C09072=1097.332,62.980,442.084,176.225,15.918,152.154
C09073=1097.327,62.731,442.101,176.223,15.918,152.154
C09074=1097.321,62.481,442.117,176.221,15.918,152.155
C09075=1097.315,62.232,442.133,176.218,15.916,152.155
C09076=1097.309,61.982,442.150,176.216,15.916,152.155
C09077=1097.304,61.733,442.167,176.213,15.915,152.156
C09078=1097.298,61.483,442.183,176.211,15.914,152.156
C09079=1097.292,61.234,442.199,176.208,15.913,152.156
C09080=1097.286,60.985,442.215,176.206,15.913,152.157
C09081=1097.280,60.735,442.232,176.204,15.912,152.157
C09082=1097.275,60.486,442.248,176.201,15.911,152.158
C09083=1097.269,60.236,442.265,176.200,15.911,152.158
C09084=1097.263,59.987,442.281,176.197,15.910,152.158
C09085=1097.257,59.738,442.297,176.195,15.909,152.158
C09086=1097.251,59.488,442.313,176.192,15.909,152.159
C09087=1097.247,59.239,442.330,176.190,15.908,152.159
C09088=1097.241,58.990,442.346,176.188,15.907,152.160
C09089=1097.235,58.741,442.362,176.185,15.906,152.160
C09090=1097.229,58.491,442.379,176.183,15.905,152.160
C09091=1097.223,58.241,442.394,176.180,15.904,152.161
C09092=1097.217,57.992,442.410,176.178,15.904,152.161
C09093=1097.212,57.742,442.427,176.176,15.903,152.161
C09094=1097.206,57.493,442.444,176.173,15.902,152.161
C09095=1097.200,57.244,442.460,176.171,15.901,152.162
C09096=1097.194,56.994,442.476,176.168,15.901,152.162
C09097=1097.188,56.745,442.492,176.167,15.900,152.162
C09098=1097.183,56.496,442.508,176.164,15.900,152.163
C09099=1097.177,56.246,442.524,176.162,15.898,152.163
C09100=1097.171,55.997,442.540,176.160,15.898,152.163
C09101=1097.166,55.747,442.557,176.157,15.897,152.164
C09102=1097.160,55.498,442.573,176.155,15.896,152.164
C09103=1097.154,55.248,442.589,176.153,15.895,152.164
C09104=1097.148,54.999,442.605,176.150,15.895,152.165
C09105=1097.143,54.750,442.621,176.148,15.894,152.165
C09106=1097.137,54.501,442.637,176.146,15.893,152.165
C09107=1097.131,54.251,442.653,176.143,15.892,152.166
C09108=1097.125,54.001,442.669,176.141,15.892,152.166
C09109=1097.119,53.752,442.685,176.139,15.890,152.166
C09110=1097.114,53.502,442.702,176.137,15.890,152.167
C09111=1097.109,53.253,442.717,176.134,15.889,152.167
C09112=1097.103,53.004,442.733,176.132,15.888,152.167
C09113=1097.097,52.754,442.750,176.130,15.887,152.167
C09114=1097.091,52.505,442.766,176.127,15.886,152.168
C09115=1097.086,52.255,442.781,176.125,15.886,152.168
C09116=1097.080,52.006,442.797,176.123,15.884,152.168
C09117=1097.074,51.757,442.814,176.120,15.884,152.169
C09118=1097.069,51.507,442.829,176.119,15.884,152.169
C09119=1097.063,51.258,442.845,176.116,15.882,152.169
C09120=1097.057,51.008,442.862,176.114,15.881,152.170
C09121=1097.052,50.759,442.877,176.111,15.880,152.170
C09122=1097.046,50.510,442.893,176.109,15.880,152.170
C09123=1097.040,50.260,442.909,176.107,15.879,152.170
C09124=1097.034,50.011,442.925,176.105,15.878,152.171
C09125=1097.029,49.762,442.941,176.103,15.877,152.171
C09126=1097.023,49.512,442.956,176.100,15.876,152.171
C09127=1097.017,49.263,442.973,176.098,15.876,152.172
C09128=1097.012,49.013,442.988,176.096,15.875,152.172
C09129=1097.006,48.764,443.004,176.093,15.874,152.172
C09130=1097.001,48.514,443.020,176.091,15.873,152.172
C09131=1096.995,48.265,443.036,176.089,15.872,152.173
C09132=1096.989,47.990,443.053,176.086,15.871,152.173
C09133=1096.982,47.715,443.071,176.084,15.870,152.173
C09134=1096.977,47.442,443.089,176.082,15.869,152.174
C09135=1096.970,47.168,443.106,176.079,15.868,152.174
C09136=1096.965,46.918,443.121,176.077,15.867,152.174
C09137=1096.959,46.668,443.137,176.074,15.867,152.175
C09138=1096.954,46.419,443.153,176.073,15.866,152.175
C09139=1096.948,46.170,443.169,176.071,15.865,152.175
C09140=1096.942,45.920,443.184,176.068,15.864,152.175
C09141=1096.937,45.671,443.200,176.066,15.863,152.176
C09142=1096.931,45.421,443.216,176.063,15.862,152.176
C09143=1096.926,45.171,443.231,176.061,15.861,152.176
C09144=1096.920,44.922,443.247,176.060,15.860,152.177
C09145=1096.915,44.672,443.263,176.057,15.859,152.177
C09146=1096.909,44.423,443.279,176.055,15.858,152.177
C09147=1096.904,44.174,443.294,176.052,15.857,152.177
C09148=1096.898,43.924,443.310,176.050,15.857,152.178
C09149=1096.891,43.675,443.325,176.048,15.856,152.178
C09150=1096.886,43.426,443.341,176.046,15.855,152.178
C09151=1096.880,43.176,443.357,176.044,15.854,152.179
C09152=1096.875,42.926,443.372,176.042,15.853,152.179
C09153=1096.870,42.677,443.388,176.039,15.852,152.179
C09154=1096.863,42.428,443.403,176.037,15.851,152.179
C09155=1096.857,42.178,443.419,176.035,15.851,152.180
C09156=1096.852,41.929,443.434,176.033,15.849,152.180
C09157=1096.846,41.679,443.450,176.031,15.849,152.180
C09158=1096.840,41.430,443.465,176.028,15.848,152.181
C09159=1096.835,41.180,443.480,176.026,15.847,152.181
C09160=1096.829,40.931,443.497,176.024,15.846,152.181
C09161=1096.823,40.681,443.512,176.021,15.845,152.181
C09162=1096.817,40.432,443.527,176.020,15.844,152.182
C09163=1096.812,40.183,443.543,176.018,15.844,152.182
C09164=1096.806,39.934,443.558,176.015,15.842,152.182
C09165=1096.801,39.684,443.574,176.013,15.842,152.182
C09166=1096.794,39.434,443.589,176.011,15.841,152.183
C09167=1096.789,39.185,443.605,176.008,15.840,152.183
C09168=1096.783,38.935,443.620,176.007,15.839,152.183
C09169=1096.778,38.686,443.635,176.005,15.838,152.183
C09170=1096.772,38.436,443.650,176.002,15.837,152.184
C09171=1096.766,38.186,443.666,176.000,15.836,152.184
C09172=1096.761,37.938,443.682,175.998,15.836,152.184
C09173=1096.755,37.688,443.697,175.996,15.834,152.184
C09174=1096.749,37.438,443.712,175.994,15.834,152.185
C09175=1096.744,37.189,443.727,175.991,15.832,152.185
C09176=1096.738,36.939,443.742,175.989,15.832,152.185
C09177=1096.732,36.691,443.758,175.987,15.831,152.186
C09178=1096.726,36.441,443.773,175.985,15.830,152.186
C09179=1096.720,36.191,443.789,175.983,15.829,152.186
C09180=1096.715,35.942,443.804,175.981,15.828,152.186
C09181=1096.709,35.692,443.819,175.978,15.827,152.187
C09182=1096.704,35.443,443.834,175.976,15.826,152.187
C09183=1096.697,35.193,443.849,175.974,15.825,152.187
C09184=1096.691,34.944,443.865,175.972,15.824,152.187
C09185=1096.686,34.695,443.880,175.970,15.823,152.188
C09186=1096.680,34.445,443.895,175.968,15.823,152.188
C09187=1096.675,34.196,443.910,175.965,15.821,152.188
C09188=1096.669,33.946,443.925,175.963,15.821,152.188
C09189=1096.664,33.697,443.941,175.961,15.820,152.189
C09190=1096.657,33.447,443.955,175.959,15.819,152.189
C09191=1096.652,33.198,443.971,175.957,15.818,152.189
C09192=1096.646,32.948,443.986,175.955,15.817,152.189
C09193=1096.640,32.698,444.001,175.952,15.816,152.190
C09194=1096.634,32.449,444.016,175.950,15.815,152.190
C09195=1096.629,32.199,444.031,175.949,15.815,152.190
C09196=1096.622,31.925,444.048,175.946,15.813,152.191
C09197=1096.616,31.651,444.064,175.944,15.813,152.191
C09198=1096.610,31.377,444.081,175.941,15.811,152.191
C09199=1096.603,31.102,444.097,175.939,15.811,152.191
C09200=1096.598,30.852,444.113,175.937,15.809,152.192
C09201=1096.592,30.603,444.128,175.935,15.809,152.192
C09202=1096.586,30.354,444.143,175.933,15.808,152.192
C09203=1096.581,30.105,444.158,175.931,15.806,152.192
C09204=1096.575,29.854,444.173,175.929,15.805,152.193
C09205=1096.569,29.605,444.187,175.927,15.805,152.193
C09206=1096.564,29.355,444.203,175.924,15.803,152.193
C09207=1096.558,29.106,444.217,175.922,15.803,152.193
C09208=1096.552,28.856,444.233,175.920,15.802,152.194
C09209=1096.547,28.607,444.247,175.918,15.801,152.194
C09210=1096.540,28.358,444.262,175.916,15.800,152.194
C09211=1096.535,28.108,444.277,175.914,15.799,152.194
C09212=1096.529,27.859,444.292,175.912,15.797,152.194
C09213=1096.523,27.610,444.307,175.910,15.797,152.195
C09214=1096.518,27.360,444.321,175.908,15.796,152.195
C09215=1096.512,27.110,444.336,175.906,15.795,152.195
C09216=1096.507,26.861,444.352,175.903,15.794,152.196
C09217=1096.500,26.611,444.367,175.901,15.793,152.196
C09218=1096.495,26.362,444.381,175.899,15.793,152.196
C09219=1096.489,26.112,444.397,175.897,15.791,152.196
C09220=1096.483,25.863,444.411,175.895,15.790,152.196
C09221=1096.477,25.613,444.425,175.893,15.789,152.197
C09222=1096.471,25.364,444.440,175.891,15.788,152.197
C09223=1096.466,25.114,444.456,175.889,15.787,152.197
C09224=1096.460,24.865,444.470,175.887,15.787,152.197
C09225=1096.454,24.615,444.484,175.885,15.786,152.198
C09226=1096.449,24.366,444.500,175.882,15.785,152.198
C09227=1096.443,24.117,444.514,175.881,15.784,152.198
C09228=1096.437,23.867,444.529,175.879,15.783,152.198
C09229=1096.432,23.618,444.544,175.876,15.782,152.199
C09230=1096.425,23.367,444.559,175.874,15.781,152.199
C09231=1096.420,23.118,444.573,175.872,15.780,152.199
C09232=1096.413,22.869,444.588,175.870,15.778,152.199
C09233=1096.409,22.619,444.602,175.868,15.778,152.200
C09234=1096.403,22.370,444.617,175.866,15.777,152.200
C09235=1096.396,22.120,444.632,175.864,15.776,152.200
C09236=1096.391,21.871,444.646,175.862,15.775,152.200
C09237=1096.385,21.621,444.661,175.860,15.774,152.200
C09238=1096.380,21.372,444.676,175.858,15.773,152.201
C09239=1096.374,21.122,444.690,175.855,15.772,152.201
C09240=1096.368,20.873,444.705,175.854,15.771,152.201
C09241=1096.363,20.623,444.720,175.852,15.770,152.201
C09242=1096.357,20.374,444.734,175.850,15.769,152.202
C09243=1096.351,20.124,444.749,175.847,15.768,152.202
C09244=1096.345,19.875,444.763,175.846,15.767,152.202
C09245=1096.339,19.625,444.778,175.844,15.766,152.202
C09246=1096.334,19.376,444.793,175.841,15.765,152.202
C09247=1096.328,19.127,444.807,175.839,15.764,152.203
C09248=1096.322,18.876,444.822,175.837,15.763,152.203
C09249=1096.316,18.627,444.836,175.836,15.763,152.203
C09250=1096.311,18.378,444.850,175.833,15.761,152.204
C09251=1096.304,18.128,444.865,175.831,15.760,152.204
C09252=1096.299,17.879,444.879,175.829,15.759,152.204
C09253=1096.293,17.629,444.894,175.828,15.759,152.204
C09254=1096.288,17.379,444.908,175.825,15.757,152.204
C09255=1096.282,17.130,444.923,175.823,15.756,152.205
C09256=1096.276,16.880,444.938,175.821,15.755,152.205
C09257=1096.270,16.631,444.952,175.820,15.755,152.205
C09258=1096.264,16.382,444.966,175.817,15.753,152.205
C09259=1096.258,16.132,444.980,175.815,15.752,152.205
C09260=1096.253,15.859,444.996,175.813,15.751,152.206
C09261=1096.246,15.586,445.012,175.811,15.750,152.206
C09262=1096.240,15.313,445.028,175.809,15.750,152.206
C09263=1096.233,15.040,445.044,175.806,15.748,152.206
C09264=1096.228,14.790,445.058,175.805,15.747,152.207
C09265=1096.222,14.542,445.072,175.803,15.746,152.207
C09266=1096.216,14.291,445.086,175.800,15.745,152.207
C09267=1096.210,14.042,445.101,175.798,15.744,152.207
C09268=1096.205,13.793,445.115,175.796,15.743,152.207
C09269=1096.199,13.542,445.129,175.795,15.743,152.208
C09270=1096.193,13.293,445.144,175.792,15.741,152.208
C09271=1096.188,13.044,445.158,175.790,15.740,152.208
C09272=1096.181,12.794,445.173,175.788,15.739,152.208
C09273=1096.176,12.545,445.186,175.787,15.739,152.209
C09274=1096.170,12.295,445.200,175.784,15.737,152.209
C09275=1096.163,12.046,445.215,175.782,15.736,152.209
C09276=1096.158,11.796,445.228,175.780,15.735,152.209
C09277=1096.152,11.547,445.243,175.779,15.735,152.210
C09278=1096.146,11.297,445.257,175.776,15.733,152.210
C09279=1096.140,11.047,445.271,175.774,15.732,152.210
C09280=1096.134,10.798,445.286,175.772,15.732,152.210
C09281=1096.129,10.549,445.300,175.770,15.731,152.210
C09282=1096.123,10.299,445.314,175.768,15.729,152.211
C09283=1096.117,10.050,445.328,175.766,15.728,152.211
C09284=1096.112,9.800,445.342,175.764,15.728,152.211
C09285=1096.105,9.550,445.356,175.763,15.726,152.211
C09286=1096.099,9.301,445.370,175.760,15.725,152.211
C09287=1096.094,9.052,445.384,175.758,15.724,152.212
C09288=1096.088,8.802,445.398,175.757,15.723,152.212
C09289=1096.082,8.552,445.412,175.755,15.723,152.212
C09290=1096.076,8.303,445.427,175.752,15.721,152.212
C09291=1096.071,8.053,445.441,175.750,15.720,152.212
C09292=1096.065,7.804,445.455,175.749,15.719,152.213
C09293=1096.059,7.554,445.468,175.747,15.719,152.213
C09294=1096.053,7.305,445.483,175.744,15.717,152.213
C09295=1096.047,7.055,445.497,175.742,15.716,152.213
C09296=1096.042,6.806,445.511,175.741,15.716,152.214
C09297=1096.036,6.556,445.525,175.739,15.714,152.214
C09298=1096.030,6.306,445.539,175.737,15.714,152.214
C09299=1096.024,6.057,445.553,175.734,15.712,152.214
C09300=1096.018,5.807,445.567,175.733,15.711,152.214
C09301=1096.013,5.558,445.580,175.731,15.710,152.215
C09302=1096.007,5.308,445.594,175.729,15.710,152.215
C09303=1096.001,5.058,445.609,175.727,15.708,152.215
C09304=1095.995,4.809,445.623,175.725,15.707,152.215
C09305=1095.989,4.560,445.636,175.723,15.706,152.215
C09306=1095.984,4.310,445.650,175.721,15.705,152.216
C09307=1095.978,4.061,445.664,175.719,15.705,152.216
C09308=1095.973,3.811,445.678,175.717,15.703,152.216
C09309=1095.967,3.561,445.692,175.715,15.702,152.216
C09310=1095.960,3.312,445.706,175.714,15.701,152.216
C09311=1095.955,3.062,445.719,175.712,15.700,152.217
C09312=1095.949,2.813,445.734,175.709,15.699,152.217
C09313=1095.944,2.563,445.748,175.707,15.698,152.217
C09314=1095.938,2.314,445.761,175.705,15.697,152.217
C09315=1095.931,2.064,445.775,175.704,15.696,152.217
C09316=1095.926,1.814,445.789,175.702,15.695,152.218
C09317=1095.921,1.565,445.803,175.700,15.694,152.218
C09318=1095.915,1.315,445.817,175.698,15.693,152.218
C09319=1095.909,1.066,445.830,175.696,15.692,152.218
C09320=1095.903,0.816,445.844,175.694,15.691,152.218
C09321=1095.898,0.567,445.858,175.692,15.690,152.219
C09322=1095.892,0.317,445.872,175.690,15.688,152.219
C09323=1095.886,0.068,445.885,175.688,15.688,152.219
C09324=1095.880,-0.203,445.900,175.687,15.687,152.219
C09325=1095.873,-0.475,445.915,175.684,15.685,152.219
C09326=1095.867,-0.746,445.931,175.682,15.685,152.220
C09327=1095.861,-1.017,445.945,175.680,15.683,152.220
C09328=1095.855,-1.266,445.959,175.678,15.682,152.220
C09329=1095.850,-1.516,445.972,175.676,15.681,152.220
C09330=1095.844,-1.765,445.986,175.674,15.680,152.220
C09331=1095.839,-2.015,446.000,175.673,15.679,152.220
C09332=1095.833,-2.264,446.013,175.671,15.678,152.221
C09333=1095.827,-2.514,446.027,175.668,15.677,152.221
C09334=1095.822,-2.763,446.041,175.666,15.676,152.221
C09335=1095.815,-3.013,446.054,175.665,15.675,152.221
C09336=1095.810,-3.262,446.068,175.663,15.674,152.221
C09337=1095.804,-3.512,446.082,175.661,15.673,152.222
C09338=1095.799,-3.762,446.095,175.659,15.672,152.222
C09339=1095.793,-4.011,446.109,175.657,15.671,152.222
C09340=1095.786,-4.261,446.122,175.655,15.670,152.222
C09341=1095.781,-4.511,446.136,175.653,15.669,152.222
C09342=1095.775,-4.760,446.149,175.652,15.668,152.223
C09343=1095.769,-5.010,446.163,175.649,15.666,152.223
C09344=1095.763,-5.259,446.176,175.647,15.666,152.223
C09345=1095.757,-5.508,446.190,175.646,15.665,152.223
C09346=1095.751,-5.758,446.203,175.644,15.664,152.223
C09347=1095.746,-6.008,446.217,175.642,15.663,152.224
C09348=1095.740,-6.257,446.230,175.640,15.662,152.224
C09349=1095.734,-6.507,446.244,175.638,15.660,152.224
C09350=1095.728,-6.756,446.257,175.636,15.660,152.224
C09351=1095.723,-7.006,446.270,175.634,15.659,152.224
C09352=1095.717,-7.255,446.284,175.633,15.658,152.225
C09353=1095.711,-7.505,446.297,175.631,15.657,152.225
C09354=1095.704,-7.755,446.311,175.628,15.655,152.225
C09355=1095.699,-8.004,446.325,175.626,15.654,152.225
C09356=1095.693,-8.254,446.337,175.625,15.653,152.225
C09357=1095.687,-8.504,446.351,175.623,15.653,152.226
C09358=1095.681,-8.753,446.365,175.621,15.651,152.226
C09359=1095.675,-9.002,446.378,175.619,15.651,152.226
C09360=1095.670,-9.253,446.391,175.617,15.649,152.226
C09361=1095.664,-9.502,446.404,175.615,15.648,152.226
C09362=1095.658,-9.751,446.418,175.613,15.648,152.227
C09363=1095.652,-10.001,446.431,175.612,15.646,152.227
C09364=1095.647,-10.251,446.445,175.610,15.646,152.227
C09365=1095.641,-10.500,446.458,175.608,15.644,152.227
C09366=1095.634,-10.749,446.471,175.606,15.643,152.227
C09367=1095.629,-11.000,446.484,175.604,15.642,152.227
C09368=1095.623,-11.249,446.498,175.602,15.641,152.228
C09369=1095.618,-11.499,446.511,175.600,15.640,152.228
C09370=1095.612,-11.748,446.524,175.599,15.639,152.228
C09371=1095.605,-11.998,446.537,175.597,15.638,152.228
C09372=1095.600,-12.247,446.551,175.595,15.638,152.228
C09373=1095.594,-12.497,446.564,175.593,15.636,152.228
C09374=1095.589,-12.746,446.577,175.591,15.635,152.229
C09375=1095.583,-12.996,446.590,175.589,15.634,152.229
C09376=1095.577,-13.245,446.603,175.587,15.633,152.229
C09377=1095.572,-13.495,446.617,175.586,15.632,152.229
C09378=1095.566,-13.745,446.629,175.584,15.631,152.229
C09379=1095.560,-13.994,446.643,175.582,15.630,152.230
C09380=1095.554,-14.244,446.656,175.580,15.629,152.230
C09381=1095.548,-14.493,446.669,175.578,15.628,152.230
C09382=1095.543,-14.743,446.683,175.576,15.627,152.230
C09383=1095.537,-14.993,446.695,175.575,15.626,152.230
C09384=1095.530,-15.242,446.709,175.573,15.625,152.231
C09385=1095.525,-15.492,446.722,175.571,15.624,152.231
C09386=1095.519,-15.742,446.735,175.568,15.623,152.231
C09387=1095.513,-15.991,446.748,175.567,15.621,152.231
C09388=1095.507,-16.260,446.762,175.565,15.621,152.231
C09389=1095.501,-16.530,446.776,175.563,15.620,152.231
C09390=1095.494,-16.799,446.790,175.561,15.618,152.232
C09391=1095.488,-17.068,446.804,175.559,15.617,152.232
C09392=1095.482,-17.318,446.817,175.557,15.616,152.232
C09393=1095.476,-17.567,446.830,175.555,15.616,152.232
C09394=1095.471,-17.817,446.843,175.554,15.615,152.232
C09395=1095.465,-18.067,446.856,175.552,15.614,152.233
C09396=1095.459,-18.316,446.869,175.549,15.612,152.233
C09397=1095.453,-18.566,446.882,175.548,15.611,152.233
C09398=1095.446,-18.815,446.895,175.546,15.610,152.233
C09399=1095.441,-19.066,446.908,175.544,15.609,152.233
C09400=1095.435,-19.315,446.922,175.543,15.608,152.234
C09401=1095.429,-19.565,446.934,175.541,15.608,152.234
C09402=1095.424,-19.813,446.947,175.539,15.606,152.234
C09403=1095.418,-20.063,446.960,175.537,15.606,152.234
C09404=1095.412,-20.313,446.972,175.535,15.604,152.234
C09405=1095.406,-20.563,446.986,175.533,15.603,152.235
C09406=1095.400,-20.812,446.999,175.531,15.602,152.235
C09407=1095.394,-21.062,447.012,175.529,15.601,152.235
C09408=1095.388,-21.312,447.024,175.528,15.600,152.235
C09409=1095.382,-21.562,447.037,175.526,15.599,152.235
C09410=1095.377,-21.810,447.050,175.524,15.598,152.235
C09411=1095.371,-22.060,447.062,175.522,15.598,152.236
C09412=1095.366,-22.310,447.076,175.521,15.596,152.236
C09413=1095.359,-22.559,447.089,175.519,15.595,152.236
C09414=1095.354,-22.809,447.101,175.517,15.594,152.236
C09415=1095.348,-23.059,447.114,175.515,15.593,152.236
C09416=1095.341,-23.308,447.127,175.513,15.592,152.236
C09417=1095.336,-23.558,447.139,175.512,15.591,152.237
C09418=1095.330,-23.808,447.152,175.510,15.590,152.237
C09419=1095.324,-24.057,447.165,175.508,15.589,152.237
C09420=1095.319,-24.307,447.178,175.506,15.588,152.237
C09421=1095.313,-24.557,447.191,175.505,15.587,152.237
C09422=1095.307,-24.806,447.204,175.502,15.586,152.238
C09423=1095.301,-25.055,447.216,175.500,15.585,152.238
C09424=1095.295,-25.305,447.229,175.498,15.584,152.238
C09425=1095.290,-25.555,447.241,175.497,15.583,152.238
C09426=1095.283,-25.804,447.255,175.495,15.582,152.238
C09427=1095.278,-26.054,447.267,175.493,15.581,152.238
C09428=1095.272,-26.303,447.279,175.492,15.580,152.238
C09429=1095.266,-26.553,447.292,175.490,15.579,152.239
C09430=1095.261,-26.803,447.306,175.488,15.578,152.239
C09431=1095.255,-27.053,447.318,175.486,15.577,152.239
C09432=1095.250,-27.302,447.331,175.484,15.575,152.239
C09433=1095.243,-27.551,447.343,175.482,15.575,152.239
C09434=1095.237,-27.801,447.355,175.481,15.574,152.240
C09435=1095.231,-28.051,447.368,175.479,15.573,152.240
C09436=1095.225,-28.301,447.381,175.477,15.572,152.240
C09437=1095.219,-28.550,447.393,175.475,15.571,152.240
C09438=1095.214,-28.800,447.406,175.474,15.570,152.240
C09439=1095.208,-29.049,447.418,175.472,15.569,152.241
C09440=1095.202,-29.299,447.431,175.470,15.568,152.241
C09441=1095.196,-29.549,447.444,175.468,15.567,152.241
C09442=1095.190,-29.799,447.457,175.467,15.566,152.241
C09443=1095.184,-30.048,447.469,175.465,15.565,152.241
C09444=1095.178,-30.298,447.481,175.463,15.564,152.241
C09445=1095.172,-30.547,447.493,175.461,15.563,152.242
C09446=1095.166,-30.797,447.506,175.459,15.562,152.242
C09447=1095.161,-31.046,447.518,175.457,15.561,152.242
C09448=1095.154,-31.295,447.531,175.455,15.560,152.242
C09449=1095.148,-31.545,447.544,175.454,15.559,152.242
C09450=1095.143,-31.795,447.556,175.452,15.558,152.242
C09451=1095.137,-32.045,447.569,175.450,15.557,152.243
C09452=1095.131,-32.313,447.582,175.449,15.556,152.243
C09453=1095.124,-32.582,447.595,175.447,15.555,152.243
C09454=1095.118,-32.850,447.609,175.444,15.554,152.243
C09455=1095.111,-33.119,447.622,175.442,15.553,152.244
C09456=1095.106,-33.368,447.634,175.441,15.552,152.244
C09457=1095.100,-33.618,447.647,175.439,15.551,152.244
C09458=1095.094,-33.868,447.659,175.437,15.550,152.244
C09459=1095.088,-34.118,447.671,175.435,15.549,152.244
C09460=1095.082,-34.367,447.684,175.434,15.548,152.244
C09461=1095.076,-34.617,447.696,175.432,15.547,152.245
C09462=1095.070,-34.866,447.709,175.430,15.546,152.245
C09463=1095.065,-35.116,447.721,175.428,15.545,152.245
C09464=1095.059,-35.366,447.733,175.427,15.544,152.245
C09465=1095.053,-35.615,447.745,175.425,15.544,152.245
C09466=1095.047,-35.865,447.758,175.423,15.542,152.245
C09467=1095.041,-36.114,447.770,175.421,15.541,152.246
C09468=1095.035,-36.364,447.783,175.419,15.540,152.246
C09469=1095.030,-36.614,447.795,175.417,15.539,152.246
C09470=1095.024,-36.863,447.807,175.416,15.538,152.246
C09471=1095.018,-37.113,447.819,175.414,15.537,152.246
C09472=1095.012,-37.363,447.832,175.412,15.536,152.247
C09473=1095.006,-37.612,447.844,175.411,15.535,152.247
C09474=1095.001,-37.862,447.856,175.409,15.534,152.247
C09475=1094.995,-38.112,447.869,175.407,15.533,152.247
C09476=1094.989,-38.361,447.880,175.405,15.532,152.247
C09477=1094.983,-38.611,447.893,175.404,15.531,152.247
C09478=1094.978,-38.860,447.905,175.402,15.530,152.248
C09479=1094.972,-39.110,447.917,175.400,15.529,152.248
C09480=1094.965,-39.360,447.929,175.398,15.529,152.248
C09481=1094.959,-39.609,447.942,175.397,15.527,152.248
C09482=1094.954,-39.859,447.954,175.395,15.527,152.248
C09483=1094.948,-40.109,447.965,175.393,15.526,152.248
C09484=1094.942,-40.359,447.978,175.391,15.525,152.249
C09485=1094.936,-40.608,447.990,175.390,15.524,152.249
C09486=1094.930,-40.857,448.002,175.388,15.523,152.249
C09487=1094.924,-41.107,448.015,175.386,15.522,152.249
C09488=1094.918,-41.356,448.026,175.384,15.521,152.249
C09489=1094.912,-41.606,448.039,175.383,15.520,152.250
C09490=1094.906,-41.857,448.051,175.381,15.519,152.250
C09491=1094.900,-42.105,448.062,175.379,15.518,152.250
C09492=1094.894,-42.355,448.075,175.377,15.517,152.250
C09493=1094.888,-42.605,448.087,175.376,15.516,152.250
C09494=1094.883,-42.855,448.098,175.374,15.516,152.250
C09495=1094.877,-43.105,448.111,175.372,15.514,152.251
C09496=1094.871,-43.353,448.122,175.370,15.514,152.251
C09497=1094.865,-43.603,448.135,175.369,15.512,152.251
C09498=1094.858,-43.853,448.147,175.367,15.512,152.251
C09499=1094.853,-44.103,448.158,175.365,15.511,152.251
C09500=1094.847,-44.353,448.171,175.364,15.510,152.252
C09501=1094.841,-44.602,448.183,175.362,15.509,152.252
C09502=1094.835,-44.851,448.195,175.360,15.508,152.252
C09503=1094.829,-45.102,448.206,175.358,15.507,152.252
C09504=1094.824,-45.351,448.218,175.357,15.506,152.252
C09505=1094.817,-45.600,448.230,175.355,15.505,152.252
C09506=1094.811,-45.851,448.242,175.353,15.504,152.253
C09507=1094.806,-46.100,448.254,175.351,15.503,152.253
C09508=1094.799,-46.350,448.266,175.350,15.502,152.253
C09509=1094.794,-46.599,448.278,175.348,15.501,152.253
C09510=1094.788,-46.849,448.290,175.346,15.501,152.253
C09511=1094.782,-47.098,448.302,175.345,15.499,152.253
C09512=1094.776,-47.348,448.313,175.343,15.499,152.254
C09513=1094.770,-47.598,448.326,175.341,15.497,152.254
C09514=1094.764,-47.847,448.337,175.339,15.497,152.254
C09515=1094.759,-48.098,448.349,175.338,15.496,152.254
C09516=1094.753,-48.365,448.362,175.336,15.495,152.254
C09517=1094.746,-48.635,448.375,175.333,15.493,152.255
C09518=1094.740,-48.904,448.387,175.331,15.492,152.255
C09519=1094.733,-49.172,448.400,175.330,15.492,152.255
C09520=1094.728,-49.422,448.412,175.328,15.491,152.255
C09521=1094.721,-49.672,448.424,175.326,15.490,152.256
C09522=1094.716,-49.921,448.436,175.324,15.489,152.256
C09523=1094.710,-50.171,448.447,175.323,15.488,152.256
C09524=1094.705,-50.420,448.459,175.321,15.487,152.256
C09525=1094.698,-50.671,448.471,175.319,15.486,152.256
C09526=1094.692,-50.920,448.483,175.318,15.485,152.256
C09527=1094.687,-51.170,448.494,175.316,15.484,152.257
C09528=1094.680,-51.419,448.506,175.314,15.483,152.257
C09529=1094.674,-51.668,448.518,175.312,15.482,152.257
C09530=1094.668,-51.919,448.530,175.310,15.482,152.257
C09531=1094.662,-52.168,448.541,175.309,15.481,152.257
C09532=1094.656,-52.418,448.552,175.307,15.480,152.258
C09533=1094.650,-52.668,448.565,175.306,15.479,152.258
C09534=1094.644,-52.917,448.576,175.304,15.479,152.258
C09535=1094.638,-53.167,448.588,175.303,15.477,152.258
C09536=1094.631,-53.417,448.599,175.301,15.477,152.258
C09537=1094.626,-53.666,448.611,175.299,15.476,152.259
C09538=1094.620,-53.916,448.622,175.297,15.475,152.259
C09539=1094.614,-54.165,448.634,175.295,15.474,152.259
C09540=1094.608,-54.416,448.646,175.294,15.473,152.259
C09541=1094.602,-54.665,448.657,175.292,15.472,152.259
C09542=1094.596,-54.915,448.669,175.290,15.472,152.260
C09543=1094.589,-55.164,448.680,175.288,15.470,152.260
C09544=1094.584,-55.414,448.692,175.286,15.470,152.260
C09545=1094.578,-55.663,448.704,175.285,15.469,152.260
C09546=1094.571,-55.913,448.715,175.283,15.468,152.260
C09547=1094.566,-56.163,448.726,175.281,15.467,152.261
C09548=1094.560,-56.413,448.738,175.279,15.466,152.261
C09549=1094.554,-56.662,448.749,175.278,15.465,152.261
C09550=1094.547,-56.912,448.761,175.276,15.464,152.261
C09551=1094.541,-57.162,448.772,175.274,15.463,152.261
C09552=1094.535,-57.411,448.784,175.273,15.463,152.261
C09553=1094.530,-57.661,448.796,175.271,15.462,152.262
C09554=1094.524,-57.911,448.807,175.269,15.461,152.262
C09555=1094.518,-58.160,448.818,175.268,15.460,152.262
C09556=1094.511,-58.410,448.830,175.266,15.460,152.262
C09557=1094.506,-58.660,448.841,175.264,15.458,152.262
C09558=1094.500,-58.909,448.853,175.263,15.458,152.263
C09559=1094.494,-59.159,448.864,175.261,15.457,152.263
C09560=1094.487,-59.408,448.876,175.259,15.456,152.263
C09561=1094.482,-59.658,448.887,175.257,15.455,152.263
C09562=1094.476,-59.908,448.899,175.256,15.454,152.263
C09563=1094.470,-60.157,448.910,175.254,15.453,152.264
C09564=1094.464,-60.407,448.921,175.252,15.453,152.264
C09565=1094.458,-60.657,448.932,175.251,15.452,152.264
C09566=1094.452,-60.907,448.944,175.249,15.451,152.264
C09567=1094.446,-61.156,448.956,175.248,15.450,152.264
C09568=1094.440,-61.406,448.967,175.246,15.449,152.264
C09569=1094.434,-61.656,448.978,175.244,15.449,152.265
C09570=1094.428,-61.905,448.989,175.242,15.448,152.265
C09571=1094.422,-62.155,449.001,175.240,15.447,152.265
C09572=1094.416,-62.404,449.012,175.239,15.446,152.265
C09573=1094.410,-62.655,449.023,175.237,15.445,152.265
C09574=1094.404,-62.904,449.035,175.235,15.444,152.266
C09575=1094.399,-63.153,449.046,175.233,15.443,152.266
C09576=1094.392,-63.403,449.057,175.231,15.443,152.266
C09577=1094.387,-63.653,449.068,175.231,15.442,152.266
C09578=1094.380,-63.903,449.080,175.229,15.441,152.266
C09579=1094.374,-64.152,449.091,175.227,15.440,152.267
C09580=1094.368,-64.423,449.103,175.225,15.439,152.267
C09581=1094.362,-64.693,449.115,175.223,15.439,152.267
C09582=1094.355,-64.963,449.127,175.222,15.438,152.267
C09583=1094.349,-65.233,449.139,175.220,15.437,152.267
C09584=1094.343,-65.483,449.151,175.218,15.436,152.268
C09585=1094.337,-65.732,449.162,175.216,15.435,152.268
C09586=1094.331,-65.982,449.173,175.214,15.434,152.268
C09587=1094.325,-66.232,449.184,175.213,15.433,152.268
C09588=1094.319,-66.481,449.195,175.211,15.432,152.268
C09589=1094.313,-66.731,449.207,175.209,15.432,152.269
C09590=1094.307,-66.980,449.218,175.208,15.431,152.269
C09591=1094.302,-67.230,449.230,175.206,15.430,152.269
C09592=1094.296,-67.480,449.241,175.205,15.429,152.269
C09593=1094.290,-67.730,449.252,175.203,15.429,152.269
C09594=1094.284,-67.979,449.263,175.201,15.428,152.270
C09595=1094.278,-68.229,449.274,175.199,15.427,152.270
C09596=1094.272,-68.479,449.285,175.198,15.426,152.270
C09597=1094.266,-68.728,449.296,175.196,15.425,152.270
C09598=1094.261,-68.978,449.306,175.194,15.424,152.270
C09599=1094.254,-69.228,449.318,175.192,15.423,152.271
C09600=1094.248,-69.477,449.329,175.191,15.423,152.271
C09601=1094.242,-69.727,449.340,175.190,15.422,152.271
C09602=1094.236,-69.977,449.351,175.188,15.421,152.271
C09603=1094.231,-70.227,449.363,175.186,15.420,152.271
C09604=1094.225,-70.476,449.374,175.184,15.420,152.272
C09605=1094.219,-70.726,449.385,175.183,15.418,152.272
C09606=1094.213,-70.976,449.396,175.181,15.418,152.272
C09607=1094.207,-71.225,449.407,175.179,15.417,152.272
C09608=1094.202,-71.475,449.418,175.178,15.417,152.272
C09609=1094.195,-71.725,449.429,175.176,15.416,152.273
C09610=1094.190,-71.974,449.440,175.175,15.415,152.273
C09611=1094.184,-72.224,449.451,175.173,15.414,152.273
C09612=1094.178,-72.473,449.462,175.171,15.413,152.273
C09613=1094.172,-72.724,449.473,175.169,15.412,152.273
C09614=1094.166,-72.973,449.484,175.167,15.411,152.274
C09615=1094.160,-73.222,449.494,175.166,15.411,152.274
C09616=1094.155,-73.472,449.505,175.165,15.410,152.274
C09617=1094.148,-73.722,449.517,175.163,15.409,152.274
C09618=1094.143,-73.972,449.527,175.161,15.408,152.274
C09619=1094.137,-74.221,449.538,175.159,15.408,152.275
C09620=1094.131,-74.471,449.549,175.158,15.406,152.275
C09621=1094.125,-74.721,449.560,175.156,15.406,152.275
C09622=1094.119,-74.970,449.571,175.155,15.406,152.275
C09623=1094.113,-75.220,449.582,175.153,15.404,152.275
C09624=1094.106,-75.470,449.593,175.151,15.404,152.275
C09625=1094.101,-75.720,449.603,175.149,15.403,152.276
C09626=1094.095,-75.969,449.614,175.148,15.402,152.276
C09627=1094.089,-76.219,449.625,175.146,15.401,152.276
C09628=1094.083,-76.469,449.636,175.145,15.401,152.276
C09629=1094.077,-76.718,449.647,175.143,15.400,152.277
C09630=1094.071,-76.968,449.658,175.141,15.399,152.277
C09631=1094.064,-77.218,449.668,175.139,15.399,152.277
C09632=1094.059,-77.467,449.679,175.137,15.398,152.277
C09633=1094.053,-77.717,449.690,175.136,15.397,152.277
C09634=1094.047,-77.967,449.700,175.135,15.397,152.278
C09635=1094.041,-78.217,449.712,175.133,15.396,152.278
C09636=1094.035,-78.467,449.723,175.131,15.395,152.278
C09637=1094.029,-78.716,449.733,175.129,15.394,152.278
C09638=1094.023,-78.965,449.744,175.127,15.393,152.278
C09639=1094.017,-79.215,449.755,175.126,15.393,152.279
C09640=1094.011,-79.465,449.766,175.125,15.392,152.279
C09641=1094.006,-79.715,449.776,175.123,15.391,152.279
C09642=1093.999,-79.964,449.786,175.121,15.391,152.279
C09643=1093.993,-80.214,449.797,175.119,15.390,152.279
C09644=1093.986,-80.486,449.809,175.117,15.389,152.280
C09645=1093.980,-80.759,449.821,175.116,15.388,152.280
C09646=1093.973,-81.032,449.832,175.114,15.388,152.280
C09647=1093.966,-81.304,449.844,175.112,15.387,152.280
C09648=1093.961,-81.553,449.855,175.111,15.387,152.281
C09649=1093.955,-81.803,449.864,175.109,15.386,152.281
C09650=1093.948,-82.053,449.876,175.107,15.385,152.281
C09651=1093.942,-82.302,449.887,175.105,15.384,152.281
C09652=1093.936,-82.552,449.897,175.103,15.384,152.282
C09653=1093.930,-82.801,449.908,175.102,15.383,152.282
C09654=1093.923,-83.052,449.918,175.101,15.382,152.282
C09655=1093.918,-83.301,449.928,175.099,15.382,152.282
C09656=1093.912,-83.551,449.939,175.097,15.381,152.282
C09657=1093.906,-83.800,449.949,175.096,15.381,152.283
C09658=1093.899,-84.051,449.960,175.094,15.380,152.283
C09659=1093.894,-84.300,449.971,175.092,15.379,152.283
C09660=1093.887,-84.549,449.981,175.090,15.378,152.283
C09661=1093.882,-84.799,449.991,175.089,15.378,152.284
C09662=1093.875,-85.049,450.002,175.087,15.378,152.284
C09663=1093.869,-85.299,450.013,175.086,15.377,152.284
C09664=1093.864,-85.549,450.023,175.084,15.376,152.284
C09665=1093.857,-85.798,450.033,175.082,15.375,152.284
C09666=1093.851,-86.048,450.044,175.081,15.375,152.285
C09667=1093.845,-86.297,450.054,175.079,15.374,152.285
C09668=1093.839,-86.548,450.065,175.077,15.374,152.285
C09669=1093.833,-86.797,450.076,175.075,15.373,152.285
C09670=1093.827,-87.047,450.086,175.074,15.372,152.286
C09671=1093.821,-87.296,450.096,175.073,15.372,152.286
C09672=1093.815,-87.545,450.107,175.071,15.371,152.286
C09673=1093.809,-87.796,450.117,175.069,15.370,152.286
C09674=1093.802,-88.045,450.128,175.067,15.370,152.287
C09675=1093.796,-88.295,450.138,175.066,15.369,152.287
C09676=1093.791,-88.545,450.149,175.064,15.368,152.287
C09677=1093.785,-88.794,450.159,175.062,15.368,152.287
C09678=1093.779,-89.044,450.169,175.060,15.367,152.287
C09679=1093.773,-89.294,450.179,175.059,15.367,152.288
C09680=1093.766,-89.544,450.191,175.057,15.366,152.288
C09681=1093.760,-89.794,450.200,175.056,15.365,152.288
C09682=1093.754,-90.043,450.211,175.054,15.364,152.288
C09683=1093.749,-90.293,450.221,175.053,15.364,152.289
C09684=1093.742,-90.542,450.231,175.051,15.364,152.289
C09685=1093.737,-90.792,450.242,175.049,15.363,152.289
C09686=1093.731,-91.042,450.252,175.047,15.362,152.289
C09687=1093.725,-91.291,450.263,175.046,15.362,152.289
C09688=1093.718,-91.542,450.273,175.044,15.361,152.290
C09689=1093.712,-91.791,450.284,175.043,15.360,152.290
C09690=1093.706,-92.041,450.293,175.041,15.360,152.290
C09691=1093.700,-92.290,450.304,175.040,15.359,152.290
C09692=1093.694,-92.540,450.314,175.038,15.359,152.291
C09693=1093.688,-92.790,450.324,175.036,15.358,152.291
C09694=1093.682,-93.039,450.334,175.034,15.357,152.291
C09695=1093.677,-93.289,450.345,175.033,15.357,152.291
C09696=1093.670,-93.539,450.354,175.031,15.356,152.292
C09697=1093.665,-93.788,450.365,175.029,15.355,152.292
C09698=1093.658,-94.039,450.375,175.028,15.355,152.292
C09699=1093.652,-94.288,450.386,175.026,15.355,152.292
C09700=1093.646,-94.538,450.396,175.025,15.354,152.292
C09701=1093.640,-94.787,450.407,175.023,15.353,152.293
C09702=1093.634,-95.037,450.416,175.022,15.353,152.293
C09703=1093.629,-95.287,450.426,175.020,15.352,152.293
C09704=1093.622,-95.537,450.437,175.018,15.351,152.293
C09705=1093.617,-95.787,450.447,175.017,15.351,152.294
C09706=1093.610,-96.036,450.457,175.015,15.351,152.294
C09707=1093.605,-96.286,450.467,175.013,15.349,152.294
C09708=1093.597,-96.561,450.479,175.011,15.349,152.294
C09709=1093.592,-96.835,450.489,175.010,15.348,152.295
C09710=1093.585,-97.109,450.500,175.008,15.347,152.295
C09711=1093.578,-97.384,450.512,175.007,15.347,152.295
C09712=1093.572,-97.634,450.522,175.005,15.347,152.295
C09713=1093.567,-97.884,450.533,175.003,15.346,152.296
C09714=1093.560,-98.133,450.542,175.001,15.345,152.296
C09715=1093.554,-98.383,450.552,175.000,15.345,152.296
C09716=1093.548,-98.633,450.563,174.998,15.345,152.296
C09717=1093.542,-98.883,450.572,174.996,15.344,152.297
C09718=1093.536,-99.132,450.582,174.995,15.344,152.297
C09719=1093.529,-99.382,450.592,174.993,15.343,152.297
C09720=1093.524,-99.632,450.603,174.991,15.342,152.297
C09721=1093.517,-99.881,450.613,174.990,15.342,152.298
C09722=1093.511,-100.131,450.622,174.988,15.342,152.298
C09723=1093.506,-100.381,450.633,174.986,15.341,152.298
C09724=1093.499,-100.631,450.643,174.985,15.341,152.298
C09725=1093.493,-100.880,450.652,174.983,15.340,152.299
C09726=1093.487,-101.130,450.663,174.981,15.340,152.299
C09727=1093.481,-101.380,450.673,174.980,15.338,152.299
C09728=1093.475,-101.629,450.682,174.979,15.338,152.299
C09729=1093.469,-101.879,450.692,174.977,15.338,152.299
C09730=1093.463,-102.129,450.702,174.975,15.337,152.300
C09731=1093.457,-102.379,450.712,174.974,15.337,152.300
C09732=1093.451,-102.628,450.722,174.972,15.336,152.300
C09733=1093.444,-102.878,450.732,174.970,15.335,152.300
C09734=1093.439,-103.128,450.742,174.969,15.335,152.301
C09735=1093.432,-103.377,450.752,174.967,15.335,152.301
C09736=1093.426,-103.627,450.762,174.965,15.334,152.301
C09737=1093.420,-103.877,450.771,174.964,15.334,152.301
C09738=1093.414,-104.126,450.782,174.962,15.333,152.302
C09739=1093.408,-104.376,450.792,174.960,15.333,152.302
C09740=1093.402,-104.626,450.801,174.959,15.332,152.302
C09741=1093.396,-104.876,450.811,174.957,15.332,152.302
C09742=1093.390,-105.126,450.821,174.955,15.331,152.303
C09743=1093.384,-105.375,450.831,174.954,15.331,152.303
C09744=1093.378,-105.625,450.841,174.952,15.330,152.303
C09745=1093.372,-105.875,450.850,174.950,15.330,152.304
C09746=1093.365,-106.125,450.860,174.949,15.330,152.304
C09747=1093.360,-106.375,450.870,174.947,15.329,152.304
C09748=1093.354,-106.624,450.880,174.945,15.328,152.304
C09749=1093.347,-106.874,450.890,174.944,15.328,152.305
C09750=1093.341,-107.123,450.899,174.942,15.327,152.305
C09751=1093.335,-107.373,450.909,174.941,15.328,152.305
C09752=1093.330,-107.623,450.919,174.939,15.327,152.305
C09753=1093.323,-107.873,450.929,174.937,15.327,152.306
C09754=1093.317,-108.122,450.939,174.936,15.326,152.306
C09755=1093.311,-108.372,450.949,174.934,15.326,152.306
C09756=1093.305,-108.622,450.958,174.932,15.325,152.306
C09757=1093.298,-108.872,450.968,174.931,15.325,152.307
C09758=1093.292,-109.122,450.977,174.929,15.324,152.307
C09759=1093.286,-109.371,450.987,174.927,15.324,152.307
C09760=1093.280,-109.621,450.996,174.926,15.324,152.307
C09761=1093.274,-109.871,451.007,174.924,15.323,152.308
C09762=1093.268,-110.120,451.017,174.923,15.323,152.308
C09763=1093.262,-110.370,451.026,174.921,15.322,152.308
C09764=1093.256,-110.620,451.036,174.919,15.322,152.309
C09765=1093.249,-110.870,451.046,174.918,15.322,152.309
C09766=1093.243,-111.120,451.055,174.916,15.321,152.309
C09767=1093.237,-111.369,451.065,174.914,15.321,152.309
C09768=1093.231,-111.619,451.074,174.913,15.320,152.310
C09769=1093.225,-111.868,451.083,174.911,15.320,152.310
C09770=1093.219,-112.118,451.093,174.910,15.320,152.310
C09771=1093.213,-112.368,451.103,174.908,15.319,152.310
C09772=1093.206,-112.634,451.114,174.906,15.318,152.311
C09773=1093.200,-112.901,451.124,174.905,15.319,152.311
C09774=1093.194,-113.167,451.134,174.903,15.318,152.311
C09775=1093.187,-113.434,451.144,174.901,15.317,152.312
C09776=1093.181,-113.683,451.154,174.899,15.317,152.312
C09777=1093.175,-113.933,451.163,174.898,15.317,152.312
C09778=1093.169,-114.183,451.173,174.896,15.316,152.312
C09779=1093.163,-114.433,451.182,174.895,15.316,152.313
C09780=1093.156,-114.682,451.192,174.893,15.316,152.313
C09781=1093.150,-114.932,451.201,174.891,15.315,152.313
C09782=1093.144,-115.182,451.211,174.890,15.315,152.313
C09783=1093.138,-115.432,451.221,174.888,15.314,152.314
C09784=1093.132,-115.682,451.230,174.887,15.314,152.314
C09785=1093.126,-115.931,451.240,174.885,15.314,152.314
C09786=1093.119,-116.181,451.249,174.883,15.313,152.315
C09787=1093.113,-116.431,451.259,174.882,15.313,152.315
C09788=1093.108,-116.680,451.268,174.880,15.313,152.315
C09789=1093.101,-116.930,451.278,174.879,15.312,152.315
C09790=1093.095,-117.180,451.287,174.877,15.312,152.316
C09791=1093.089,-117.429,451.297,174.876,15.312,152.316
C09792=1093.083,-117.679,451.306,174.873,15.312,152.316
C09793=1093.077,-117.929,451.316,174.872,15.311,152.317
C09794=1093.070,-118.179,451.325,174.870,15.311,152.317
C09795=1093.064,-118.429,451.334,174.869,15.310,152.317
C09796=1093.058,-118.679,451.343,174.867,15.310,152.317
C09797=1093.052,-118.929,451.353,174.865,15.310,152.318
C09798=1093.046,-119.178,451.362,174.863,15.309,152.318
C09799=1093.040,-119.427,451.372,174.862,15.309,152.318
C09800=1093.034,-119.677,451.381,174.860,15.308,152.318
C09801=1093.028,-119.927,451.391,174.859,15.309,152.319
C09802=1093.021,-120.177,451.400,174.857,15.308,152.319
C09803=1093.015,-120.427,451.410,174.856,15.308,152.319
C09804=1093.009,-120.677,451.418,174.854,15.307,152.320
C09805=1093.002,-120.927,451.428,174.852,15.307,152.320
C09806=1092.997,-121.176,451.437,174.851,15.307,152.320
C09807=1092.991,-121.425,451.446,174.849,15.307,152.321
C09808=1092.985,-121.675,451.456,174.848,15.306,152.321
C09809=1092.978,-121.925,451.466,174.846,15.306,152.321
C09810=1092.972,-122.175,451.475,174.844,15.306,152.321
C09811=1092.966,-122.425,451.483,174.843,15.306,152.322
C09812=1092.959,-122.675,451.493,174.841,15.305,152.322
C09813=1092.954,-122.924,451.502,174.840,15.305,152.322
C09814=1092.948,-123.174,451.512,174.837,15.305,152.323
C09815=1092.942,-123.423,451.521,174.836,15.304,152.323
C09816=1092.936,-123.674,451.530,174.834,15.304,152.323
C09817=1092.929,-123.923,451.539,174.833,15.304,152.323
C09818=1092.923,-124.173,451.549,174.831,15.304,152.324
C09819=1092.917,-124.422,451.558,174.830,15.303,152.324
C09820=1092.911,-124.672,451.567,174.828,15.303,152.324
C09821=1092.905,-124.922,451.576,174.827,15.303,152.324
C09822=1092.898,-125.172,451.585,174.825,15.303,152.325
C09823=1092.892,-125.422,451.595,174.824,15.302,152.325
C09824=1092.886,-125.672,451.604,174.822,15.302,152.325
C09825=1092.880,-125.921,451.613,174.819,15.302,152.326
C09826=1092.874,-126.171,451.622,174.818,15.302,152.326
C09827=1092.867,-126.421,451.631,174.816,15.301,152.326
C09828=1092.861,-126.670,451.641,174.815,15.301,152.327
C09829=1092.855,-126.921,451.650,174.813,15.301,152.327
C09830=1092.848,-127.170,451.659,174.812,15.301,152.327
C09831=1092.843,-127.419,451.668,174.810,15.300,152.328
C09832=1092.836,-127.680,451.678,174.809,15.300,152.328
C09833=1092.830,-127.939,451.688,174.807,15.300,152.328
C09834=1092.824,-128.199,451.697,174.806,15.300,152.328
C09835=1092.828,-128.456,451.709,174.804,15.296,152.328
C09836=1092.422,-128.478,451.594,174.760,15.405,152.358
C09837=1092.418,-128.220,451.581,174.761,15.408,152.359
C09838=1092.422,-127.961,451.571,174.763,15.409,152.358
C09839=1092.429,-127.702,451.562,174.764,15.409,152.358
C09840=1092.435,-127.442,451.552,174.766,15.409,152.358
C09841=1092.441,-127.192,451.543,174.768,15.409,152.357
C09842=1092.447,-126.942,451.534,174.769,15.410,152.357
C09843=1092.454,-126.693,451.525,174.771,15.410,152.357
C09844=1092.460,-126.442,451.516,174.772,15.410,152.357
C09845=1092.466,-126.192,451.506,174.774,15.410,152.356
C09846=1092.472,-125.943,451.497,174.775,15.411,152.356
C09847=1092.479,-125.694,451.488,174.777,15.411,152.356
C09848=1092.485,-125.443,451.479,174.779,15.411,152.355
C09849=1092.491,-125.194,451.470,174.781,15.411,152.355
C09850=1092.497,-124.944,451.460,174.782,15.412,152.355
C09851=1092.504,-124.694,451.451,174.784,15.412,152.355
C09852=1092.509,-124.445,451.442,174.786,15.412,152.354
C09853=1092.515,-124.195,451.433,174.787,15.412,152.354
C09854=1092.521,-123.945,451.423,174.789,15.413,152.354
C09855=1092.528,-123.695,451.414,174.790,15.413,152.353
C09856=1092.535,-123.446,451.405,174.792,15.413,152.353
C09857=1092.540,-123.195,451.396,174.793,15.413,152.353
C09858=1092.546,-122.946,451.387,174.795,15.414,152.353
C09859=1092.552,-122.696,451.377,174.796,15.414,152.352
C09860=1092.558,-122.447,451.368,174.798,15.414,152.352
C09861=1092.565,-122.197,451.358,174.800,15.415,152.352
C09862=1092.571,-121.947,451.349,174.801,15.415,152.351
C09863=1092.577,-121.697,451.340,174.803,15.416,152.351
C09864=1092.583,-121.448,451.331,174.804,15.416,152.351
C09865=1092.589,-121.198,451.322,174.807,15.416,152.351
C09866=1092.595,-120.948,451.312,174.808,15.416,152.350
C09867=1092.601,-120.698,451.302,174.810,15.417,152.350
C09868=1092.608,-120.449,451.293,174.811,15.417,152.350
C09869=1092.614,-120.199,451.283,174.813,15.417,152.350
C09870=1092.620,-119.949,451.275,174.815,15.418,152.349
C09871=1092.626,-119.699,451.265,174.816,15.418,152.349
C09872=1092.632,-119.450,451.256,174.818,15.418,152.349
C09873=1092.638,-119.200,451.247,174.820,15.419,152.348
C09874=1092.644,-118.950,451.237,174.821,15.419,152.348
C09875=1092.651,-118.700,451.228,174.823,15.420,152.348
C09876=1092.657,-118.451,451.218,174.824,15.419,152.348
C09877=1092.663,-118.201,451.208,174.826,15.420,152.347
C09878=1092.669,-117.951,451.199,174.827,15.420,152.347
C09879=1092.675,-117.701,451.189,174.829,15.421,152.347
C09880=1092.681,-117.451,451.180,174.831,15.421,152.346
C09881=1092.687,-117.202,451.171,174.832,15.422,152.346
C09882=1092.694,-116.952,451.162,174.834,15.422,152.346
C09883=1092.700,-116.702,451.153,174.835,15.422,152.346
C09884=1092.706,-116.453,451.143,174.837,15.422,152.345
C09885=1092.712,-116.203,451.134,174.839,15.423,152.345
C09886=1092.718,-115.953,451.124,174.840,15.423,152.345
C09887=1092.724,-115.703,451.114,174.842,15.424,152.345
C09888=1092.731,-115.453,451.105,174.843,15.424,152.344
C09889=1092.737,-115.204,451.095,174.845,15.425,152.344
C09890=1092.743,-114.954,451.086,174.847,15.425,152.344
C09891=1092.749,-114.704,451.076,174.848,15.425,152.343
C09892=1092.755,-114.455,451.067,174.850,15.426,152.343
C09893=1092.761,-114.205,451.057,174.851,15.426,152.343
C09894=1092.767,-113.955,451.048,174.853,15.426,152.343
C09895=1092.773,-113.706,451.038,174.855,15.427,152.342
C09896=1092.779,-113.456,451.029,174.856,15.427,152.342
C09897=1092.786,-113.189,451.018,174.858,15.428,152.342
C09898=1092.792,-112.922,451.008,174.860,15.428,152.342
C09899=1092.799,-112.655,450.997,174.862,15.429,152.341
C09900=1092.805,-112.389,450.988,174.863,15.429,152.341
C09901=1092.812,-112.139,450.978,174.865,15.429,152.341
C09902=1092.817,-111.889,450.968,174.867,15.430,152.340
C09903=1092.823,-111.639,450.958,174.868,15.430,152.340
C09904=1092.829,-111.389,450.949,174.870,15.431,152.340
C09905=1092.836,-111.140,450.939,174.871,15.431,152.340
C09906=1092.842,-110.890,450.930,174.873,15.431,152.339
C09907=1092.848,-110.640,450.920,174.875,15.432,152.339
C09908=1092.854,-110.391,450.910,174.876,15.432,152.339
C09909=1092.861,-110.141,450.900,174.878,15.433,152.339
C09910=1092.867,-109.891,450.891,174.880,15.434,152.338
C09911=1092.873,-109.641,450.881,174.881,15.434,152.338
C09912=1092.879,-109.392,450.872,174.883,15.434,152.338
C09913=1092.885,-109.142,450.862,174.884,15.434,152.338
C09914=1092.891,-108.892,450.852,174.886,15.435,152.337
C09915=1092.897,-108.642,450.842,174.888,15.436,152.337
C09916=1092.903,-108.392,450.833,174.889,15.436,152.337
C09917=1092.910,-108.143,450.822,174.891,15.436,152.337
C09918=1092.916,-107.893,450.813,174.893,15.437,152.336
C09919=1092.922,-107.643,450.803,174.894,15.437,152.336
C09920=1092.928,-107.394,450.794,174.896,15.438,152.336
C09921=1092.934,-107.144,450.784,174.898,15.439,152.336
C09922=1092.940,-106.894,450.774,174.899,15.439,152.335
C09923=1092.946,-106.644,450.764,174.901,15.439,152.335
C09924=1092.952,-106.395,450.754,174.903,15.440,152.335
C09925=1092.958,-106.145,450.745,174.904,15.440,152.335
C09926=1092.965,-105.895,450.735,174.906,15.441,152.334
C09927=1092.970,-105.645,450.725,174.908,15.441,152.334
C09928=1092.977,-105.396,450.715,174.909,15.441,152.334
C09929=1092.983,-105.146,450.705,174.911,15.442,152.334
C09930=1092.989,-104.896,450.695,174.913,15.443,152.333
C09931=1092.995,-104.646,450.686,174.914,15.443,152.333
C09932=1093.001,-104.396,450.676,174.916,15.444,152.333
C09933=1093.007,-104.147,450.665,174.917,15.444,152.333
C09934=1093.013,-103.897,450.656,174.919,15.444,152.332
C09935=1093.019,-103.648,450.646,174.920,15.445,152.332
C09936=1093.025,-103.397,450.636,174.922,15.446,152.332
C09937=1093.031,-103.148,450.626,174.923,15.446,152.332
C09938=1093.037,-102.898,450.616,174.925,15.446,152.331
C09939=1093.044,-102.649,450.607,174.927,15.448,152.331
C09940=1093.049,-102.399,450.596,174.928,15.448,152.331
C09941=1093.055,-102.149,450.586,174.930,15.448,152.331
C09942=1093.062,-101.900,450.577,174.932,15.449,152.331
C09943=1093.067,-101.649,450.566,174.933,15.449,152.330
C09944=1093.074,-101.400,450.556,174.935,15.450,152.330
C09945=1093.080,-101.150,450.547,174.937,15.450,152.330
C09946=1093.086,-100.901,450.537,174.939,15.451,152.330
C09947=1093.092,-100.651,450.526,174.940,15.451,152.329
C09948=1093.098,-100.401,450.517,174.942,15.452,152.329
C09949=1093.104,-100.152,450.507,174.944,15.453,152.329
C09950=1093.110,-99.902,450.496,174.945,15.453,152.329
C09951=1093.116,-99.652,450.487,174.947,15.453,152.328
C09952=1093.122,-99.402,450.477,174.948,15.454,152.328
C09953=1093.129,-99.153,450.467,174.949,15.455,152.328
C09954=1093.134,-98.903,450.457,174.951,15.455,152.328
C09955=1093.140,-98.653,450.447,174.953,15.456,152.327
C09956=1093.147,-98.404,450.436,174.954,15.456,152.327
C09957=1093.153,-98.153,450.426,174.956,15.457,152.327
C09958=1093.159,-97.904,450.416,174.958,15.457,152.327
C09959=1093.165,-97.654,450.406,174.960,15.458,152.326
C09960=1093.171,-97.404,450.396,174.961,15.458,152.326
C09961=1093.177,-97.130,450.385,174.963,15.459,152.326
C09962=1093.184,-96.855,450.373,174.964,15.460,152.326
C09963=1093.191,-96.580,450.363,174.966,15.461,152.326
C09964=1093.197,-96.306,450.351,174.968,15.461,152.325
C09965=1093.203,-96.056,450.342,174.970,15.462,152.325
C09966=1093.209,-95.807,450.331,174.971,15.462,152.325
C09967=1093.215,-95.557,450.321,174.973,15.463,152.324
C09968=1093.221,-95.307,450.311,174.975,15.464,152.324
C09969=1093.227,-95.058,450.301,174.977,15.465,152.324
C09970=1093.233,-94.807,450.291,174.978,15.465,152.324
C09971=1093.240,-94.558,450.280,174.980,15.465,152.324
C09972=1093.245,-94.307,450.270,174.981,15.466,152.323
C09973=1093.252,-94.058,450.260,174.982,15.467,152.323
C09974=1093.257,-93.808,450.249,174.984,15.467,152.323
C09975=1093.263,-93.559,450.239,174.986,15.468,152.323
C09976=1093.269,-93.309,450.229,174.988,15.469,152.323
C09977=1093.275,-93.060,450.219,174.989,15.469,152.322
C09978=1093.281,-92.810,450.209,174.991,15.470,152.322
C09979=1093.287,-92.560,450.198,174.993,15.471,152.322
C09980=1093.293,-92.310,450.188,174.994,15.471,152.322
C09981=1093.298,-92.061,450.177,174.996,15.471,152.321
C09982=1093.305,-91.811,450.168,174.997,15.472,152.321
C09983=1093.311,-91.561,450.156,174.999,15.473,152.321
C09984=1093.317,-91.311,450.147,175.001,15.474,152.321
C09985=1093.323,-91.062,450.136,175.002,15.474,152.321
C09986=1093.329,-90.812,450.126,175.004,15.475,152.320
C09987=1093.335,-90.562,450.116,175.006,15.476,152.320
C09988=1093.341,-90.312,450.106,175.007,15.476,152.320
C09989=1093.347,-90.063,450.095,175.009,15.476,152.320
C09990=1093.353,-89.814,450.085,175.010,15.477,152.319
C09991=1093.359,-89.563,450.074,175.012,15.478,152.319
C09992=1093.366,-89.314,450.064,175.014,15.479,152.319
C09993=1093.371,-89.064,450.054,175.015,15.479,152.319
C09994=1093.377,-88.814,450.043,175.017,15.480,152.319
C09995=1093.383,-88.565,450.033,175.019,15.480,152.318
C09996=1093.389,-88.315,450.023,175.020,15.482,152.318
//INST
///DATE 2021/06/25 14:44
///ATTR SC,RW,RJ
////FRAME ROBOT
///GROUP1 RB1
NOP
MOVL C00000 V=800.0 PL=0
MOVL C00001 V=800.0 PL=0
MOVL C00002 V=800.0 PL=0
MOVL C00003 V=800.0 PL=0
MOVL C00004 V=800.0 PL=0
MOVL C00005 V=800.0 PL=0
MOVL C00006 V=800.0 PL=0
MOVL C00007 V=800.0 PL=0
MOVL C00008 V=800.0 PL=0
MOVL C00009 V=800.0 PL=0
MOVL C00010 V=800.0 PL=0
MOVL C00011 V=800.0 PL=0
MOVL C00012 V=800.0 PL=0
MOVL C00013 V=800.0 PL=0
MOVL C00014 V=800.0 PL=0
MOVL C00015 V=800.0 PL=0
MOVL C00016 V=800.0 PL=0
MOVL C00017 V=800.0 PL=0
MOVL C00018 V=800.0 PL=0
MOVL C00019 V=800.0 PL=0
MOVL C00020 V=800.0 PL=0
MOVL C00021 V=800.0 PL=0
MOVL C00022 V=800.0 PL=0
MOVL C00023 V=800.0 PL=0
MOVL C00024 V=800.0 PL=0
MOVL C00025 V=800.0 PL=0
MOVL C00026 V=800.0 PL=0
MOVL C00027 V=800.0 PL=0
MOVL C00028 V=800.0 PL=0
MOVL C00029 V=800.0 PL=0
MOVL C00030 V=800.0 PL=0
MOVL C00031 V=800.0 PL=0
MOVL C00032 V=800.0 PL=0
MOVL C00033 V=800.0 PL=0
MOVL C00034 V=800.0 PL=0
MOVL C00035 V=800.0 PL=0
MOVL C00036 V=800.0 PL=0
MOVL C00037 V=800.0 PL=0
MOVL C00038 V=800.0 PL=0
MOVL C00039 V=800.0 PL=0
MOVL C00040 V=800.0 PL=0
MOVL C00041 V=800.0 PL=0
MOVL C00042 V=800.0 PL=0
MOVL C00043 V=800.0 PL=0
MOVL C00044 V=800.0 PL=0
MOVL C00045 V=800.0 PL=0
MOVL C00046 V=800.0 PL=0
MOVL C00047 V=800.0 PL=0
MOVL C00048 V=800.0 PL=0
MOVL C00049 V=800.0 PL=0
MOVL C00050 V=800.0 PL=0
MOVL C00051 V=800.0 PL=0
MOVL C00052 V=800.0 PL=0
MOVL C00053 V=800.0 PL=0
MOVL C00054 V=800.0 PL=0
MOVL C00055 V=800.0 PL=0
MOVL C00056 V=800.0 PL=0
MOVL C00057 V=800.0 PL=0
MOVL C00058 V=800.0 PL=0
MOVL C00059 V=800.0 PL=0
MOVL C00060 V=800.0 PL=0
MOVL C00061 V=800.0 PL=0
MOVL C00062 V=800.0 PL=0
MOVL C00063 V=800.0 PL=0
MOVL C00064 V=800.0 PL=0
MOVL C00065 V=800.0 PL=0
MOVL C00066 V=800.0 PL=0
MOVL C00067 V=800.0 PL=0
MOVL C00068 V=800.0 PL=0
MOVL C00069 V=800.0 PL=0
MOVL C00070 V=800.0 PL=0
MOVL C00071 V=800.0 PL=0
MOVL C00072 V=800.0 PL=0
MOVL C00073 V=800.0 PL=0
MOVL C00074 V=800.0 PL=0
MOVL C00075 V=800.0 PL=0
MOVL C00076 V=800.0 PL=0
MOVL C00077 V=800.0 PL=0
MOVL C00078 V=800.0 PL=0
MOVL C00079 V=800.0 PL=0
MOVL C00080 V=800.0 PL=0
MOVL C00081 V=800.0 PL=0
MOVL C00082 V=800.0 PL=0
MOVL C00083 V=800.0 PL=0
MOVL C00084 V=800.0 PL=0
MOVL C00085 V=800.0 PL=0
MOVL C00086 V=800.0 PL=0
MOVL C00087 V=800.0 PL=0
MOVL C00088 V=800.0 PL=0
MOVL C00089 V=800.0 PL=0
MOVL C00090 V=800.0 PL=0
MOVL C00091 V=800.0 PL=0
MOVL C00092 V=800.0 PL=0
MOVL C00093 V=800.0 PL=0
MOVL C00094 V=800.0 PL=0
MOVL C00095 V=800.0 PL=0
MOVL C00096 V=800.0 PL=0
MOVL C00097 V=800.0 PL=0
MOVL C00098 V=800.0 PL=0
MOVL C00099 V=800.0 PL=0
MOVL C00100 V=800.0 PL=0
MOVL C00101 V=800.0 PL=0
MOVL C00102 V=800.0 PL=0
MOVL C00103 V=800.0 PL=0
MOVL C00104 V=800.0 PL=0
MOVL C00105 V=800.0 PL=0
MOVL C00106 V=800.0 PL=0
MOVL C00107 V=800.0 PL=0
MOVL C00108 V=800.0 PL=0
MOVL C00109 V=800.0 PL=0
MOVL C00110 V=800.0 PL=0
MOVL C00111 V=800.0 PL=0
MOVL C00112 V=800.0 PL=0
MOVL C00113 V=800.0 PL=0
MOVL C00114 V=800.0 PL=0
MOVL C00115 V=800.0 PL=0
MOVL C00116 V=800.0 PL=0
MOVL C00117 V=800.0 PL=0
MOVL C00118 V=800.0 PL=0
MOVL C00119 V=800.0 PL=0
MOVL C00120 V=800.0 PL=0
MOVL C00121 V=800.0 PL=0
MOVL C00122 V=800.0 PL=0
MOVL C00123 V=800.0 PL=0
MOVL C00124 V=800.0 PL=0
MOVL C00125 V=800.0 PL=0
MOVL C00126 V=800.0 PL=0
MOVL C00127 V=800.0 PL=0
MOVL C00128 V=800.0 PL=0
MOVL C00129 V=800.0 PL=0
MOVL C00130 V=800.0 PL=0
MOVL C00131 V=800.0 PL=0
MOVL C00132 V=800.0 PL=0
MOVL C00133 V=800.0 PL=0
MOVL C00134 V=800.0 PL=0
MOVL C00135 V=800.0 PL=0
MOVL C00136 V=800.0 PL=0
MOVL C00137 V=800.0 PL=0
MOVL C00138 V=800.0 PL=0
MOVL C00139 V=800.0 PL=0
MOVL C00140 V=800.0 PL=0
MOVL C00141 V=800.0 PL=0
MOVL C00142 V=800.0 PL=0
MOVL C00143 V=800.0 PL=0
MOVL C00144 V=800.0 PL=0
MOVL C00145 V=800.0 PL=0
MOVL C00146 V=800.0 PL=0
MOVL C00147 V=800.0 PL=0
MOVL C00148 V=800.0 PL=0
MOVL C00149 V=800.0 PL=0
MOVL C00150 V=800.0 PL=0
MOVL C00151 V=800.0 PL=0
MOVL C00152 V=800.0 PL=0
MOVL C00153 V=800.0 PL=0
MOVL C00154 V=800.0 PL=0
MOVL C00155 V=800.0 PL=0
MOVL C00156 V=800.0 PL=0
MOVL C00157 V=800.0 PL=0
MOVL C00158 V=800.0 PL=0
MOVL C00159 V=800.0 PL=0
MOVL C00160 V=800.0 PL=0
MOVL C00161 V=800.0 PL=0
MOVL C00162 V=800.0 PL=0
MOVL C00163 V=800.0 PL=0
MOVL C00164 V=800.0 PL=0
MOVL C00165 V=800.0 PL=0
MOVL C00166 V=800.0 PL=0
MOVL C00167 V=800.0 PL=0
MOVL C00168 V=800.0 PL=0
MOVL C00169 V=800.0 PL=0
MOVL C00170 V=800.0 PL=0
MOVL C00171 V=800.0 PL=0
MOVL C00172 V=800.0 PL=0
MOVL C00173 V=800.0 PL=0
MOVL C00174 V=800.0 PL=0
MOVL C00175 V=800.0 PL=0
MOVL C00176 V=800.0 PL=0
MOVL C00177 V=800.0 PL=0
MOVL C00178 V=800.0 PL=0
MOVL C00179 V=800.0 PL=0
MOVL C00180 V=800.0 PL=0
MOVL C00181 V=800.0 PL=0
MOVL C00182 V=800.0 PL=0
MOVL C00183 V=800.0 PL=0
MOVL C00184 V=800.0 PL=0
MOVL C00185 V=800.0 PL=0
MOVL C00186 V=800.0 PL=0
MOVL C00187 V=800.0 PL=0
MOVL C00188 V=800.0 PL=0
MOVL C00189 V=800.0 PL=0
MOVL C00190 V=800.0 PL=0
MOVL C00191 V=800.0 PL=0
MOVL C00192 V=800.0 PL=0
MOVL C00193 V=800.0 PL=0
MOVL C00194 V=800.0 PL=0
MOVL C00195 V=800.0 PL=0
MOVL C00196 V=800.0 PL=0
MOVL C00197 V=800.0 PL=0
MOVL C00198 V=800.0 PL=0
MOVL C00199 V=800.0 PL=0
MOVL C00200 V=800.0 PL=0
MOVL C00201 V=800.0 PL=0
MOVL C00202 V=800.0 PL=0
MOVL C00203 V=800.0 PL=0
MOVL C00204 V=800.0 PL=0
MOVL C00205 V=800.0 PL=0
MOVL C00206 V=800.0 PL=0
MOVL C00207 V=800.0 PL=0
MOVL C00208 V=800.0 PL=0
MOVL C00209 V=800.0 PL=0
MOVL C00210 V=800.0 PL=0
MOVL C00211 V=800.0 PL=0
MOVL C00212 V=800.0 PL=0
MOVL C00213 V=800.0 PL=0
MOVL C00214 V=800.0 PL=0
MOVL C00215 V=800.0 PL=0
MOVL C00216 V=800.0 PL=0
MOVL C00217 V=800.0 PL=0
MOVL C00218 V=800.0 PL=0
MOVL C00219 V=800.0 PL=0
MOVL C00220 V=800.0 PL=0
MOVL C00221 V=800.0 PL=0
MOVL C00222 V=800.0 PL=0
MOVL C00223 V=800.0 PL=0
MOVL C00224 V=800.0 PL=0
MOVL C00225 V=800.0 PL=0
MOVL C00226 V=800.0 PL=0
MOVL C00227 V=800.0 PL=0
MOVL C00228 V=800.0 PL=0
MOVL C00229 V=800.0 PL=0
MOVL C00230 V=800.0 PL=0
MOVL C00231 V=800.0 PL=0
MOVL C00232 V=800.0 PL=0
MOVL C00233 V=800.0 PL=0
MOVL C00234 V=800.0 PL=0
MOVL C00235 V=800.0 PL=0
MOVL C00236 V=800.0 PL=0
MOVL C00237 V=800.0 PL=0
MOVL C00238 V=800.0 PL=0
MOVL C00239 V=800.0 PL=0
MOVL C00240 V=800.0 PL=0
MOVL C00241 V=800.0 PL=0
MOVL C00242 V=800.0 PL=0
MOVL C00243 V=800.0 PL=0
MOVL C00244 V=800.0 PL=0
MOVL C00245 V=800.0 PL=0
MOVL C00246 V=800.0 PL=0
MOVL C00247 V=800.0 PL=0
MOVL C00248 V=800.0 PL=0
MOVL C00249 V=800.0 PL=0
MOVL C00250 V=800.0 PL=0
MOVL C00251 V=800.0 PL=0
MOVL C00252 V=800.0 PL=0
MOVL C00253 V=800.0 PL=0
MOVL C00254 V=800.0 PL=0
MOVL C00255 V=800.0 PL=0
MOVL C00256 V=800.0 PL=0
MOVL C00257 V=800.0 PL=0
MOVL C00258 V=800.0 PL=0
MOVL C00259 V=800.0 PL=0
MOVL C00260 V=800.0 PL=0
MOVL C00261 V=800.0 PL=0
MOVL C00262 V=800.0 PL=0
MOVL C00263 V=800.0 PL=0
MOVL C00264 V=800.0 PL=0
MOVL C00265 V=800.0 PL=0
MOVL C00266 V=800.0 PL=0
MOVL C00267 V=800.0 PL=0
MOVL C00268 V=800.0 PL=0
MOVL C00269 V=800.0 PL=0
MOVL C00270 V=800.0 PL=0
MOVL C00271 V=800.0 PL=0
MOVL C00272 V=800.0 PL=0
MOVL C00273 V=800.0 PL=0
MOVL C00274 V=800.0 PL=0
MOVL C00275 V=800.0 PL=0
MOVL C00276 V=800.0 PL=0
MOVL C00277 V=800.0 PL=0
MOVL C00278 V=800.0 PL=0
MOVL C00279 V=800.0 PL=0
MOVL C00280 V=800.0 PL=0
MOVL C00281 V=800.0 PL=0
MOVL C00282 V=800.0 PL=0
MOVL C00283 V=800.0 PL=0
MOVL C00284 V=800.0 PL=0
MOVL C00285 V=800.0 PL=0
MOVL C00286 V=800.0 PL=0
MOVL C00287 V=800.0 PL=0
MOVL C00288 V=800.0 PL=0
MOVL C00289 V=800.0 PL=0
MOVL C00290 V=800.0 PL=0
MOVL C00291 V=800.0 PL=0
MOVL C00292 V=800.0 PL=0
MOVL C00293 V=800.0 PL=0
MOVL C00294 V=800.0 PL=0
MOVL C00295 V=800.0 PL=0
MOVL C00296 V=800.0 PL=0
MOVL C00297 V=800.0 PL=0
MOVL C00298 V=800.0 PL=0
MOVL C00299 V=800.0 PL=0
MOVL C00300 V=800.0 PL=0
MOVL C00301 V=800.0 PL=0
MOVL C00302 V=800.0 PL=0
MOVL C00303 V=800.0 PL=0
MOVL C00304 V=800.0 PL=0
MOVL C00305 V=800.0 PL=0
MOVL C00306 V=800.0 PL=0
MOVL C00307 V=800.0 PL=0
MOVL C00308 V=800.0 PL=0
MOVL C00309 V=800.0 PL=0
MOVL C00310 V=800.0 PL=0
MOVL C00311 V=800.0 PL=0
MOVL C00312 V=800.0 PL=0
MOVL C00313 V=800.0 PL=0
MOVL C00314 V=800.0 PL=0
MOVL C00315 V=800.0 PL=0
MOVL C00316 V=800.0 PL=0
MOVL C00317 V=800.0 PL=0
MOVL C00318 V=800.0 PL=0
MOVL C00319 V=800.0 PL=0
MOVL C00320 V=800.0 PL=0
MOVL C00321 V=800.0 PL=0
MOVL C00322 V=800.0 PL=0
MOVL C00323 V=800.0 PL=0
MOVL C00324 V=800.0 PL=0
MOVL C00325 V=800.0 PL=0
MOVL C00326 V=800.0 PL=0
MOVL C00327 V=800.0 PL=0
MOVL C00328 V=800.0 PL=0
MOVL C00329 V=800.0 PL=0
MOVL C00330 V=800.0 PL=0
MOVL C00331 V=800.0 PL=0
MOVL C00332 V=800.0 PL=0
MOVL C00333 V=800.0 PL=0
MOVL C00334 V=800.0 PL=0
MOVL C00335 V=800.0 PL=0
MOVL C00336 V=800.0 PL=0
MOVL C00337 V=800.0 PL=0
MOVL C00338 V=800.0 PL=0
MOVL C00339 V=800.0 PL=0
MOVL C00340 V=800.0 PL=0
MOVL C00341 V=800.0 PL=0
MOVL C00342 V=800.0 PL=0
MOVL C00343 V=800.0 PL=0
MOVL C00344 V=800.0 PL=0
MOVL C00345 V=800.0 PL=0
MOVL C00346 V=800.0 PL=0
MOVL C00347 V=800.0 PL=0
MOVL C00348 V=800.0 PL=0
MOVL C00349 V=800.0 PL=0
MOVL C00350 V=800.0 PL=0
MOVL C00351 V=800.0 PL=0
MOVL C00352 V=800.0 PL=0
MOVL C00353 V=800.0 PL=0
MOVL C00354 V=800.0 PL=0
MOVL C00355 V=800.0 PL=0
MOVL C00356 V=800.0 PL=0
MOVL C00357 V=800.0 PL=0
MOVL C00358 V=800.0 PL=0
MOVL C00359 V=800.0 PL=0
MOVL C00360 V=800.0 PL=0
MOVL C00361 V=800.0 PL=0
MOVL C00362 V=800.0 PL=0
MOVL C00363 V=800.0 PL=0
MOVL C00364 V=800.0 PL=0
MOVL C00365 V=800.0 PL=0
MOVL C00366 V=800.0 PL=0
MOVL C00367 V=800.0 PL=0
MOVL C00368 V=800.0 PL=0
MOVL C00369 V=800.0 PL=0
MOVL C00370 V=800.0 PL=0
MOVL C00371 V=800.0 PL=0
MOVL C00372 V=800.0 PL=0
MOVL C00373 V=800.0 PL=0
MOVL C00374 V=800.0 PL=0
MOVL C00375 V=800.0 PL=0
MOVL C00376 V=800.0 PL=0
MOVL C00377 V=800.0 PL=0
MOVL C00378 V=800.0 PL=0
MOVL C00379 V=800.0 PL=0
MOVL C00380 V=800.0 PL=0
MOVL C00381 V=800.0 PL=0
MOVL C00382 V=800.0 PL=0
MOVL C00383 V=800.0 PL=0
MOVL C00384 V=800.0 PL=0
MOVL C00385 V=800.0 PL=0
MOVL C00386 V=800.0 PL=0
MOVL C00387 V=800.0 PL=0
MOVL C00388 V=800.0 PL=0
MOVL C00389 V=800.0 PL=0
MOVL C00390 V=800.0 PL=0
MOVL C00391 V=800.0 PL=0
MOVL C00392 V=800.0 PL=0
MOVL C00393 V=800.0 PL=0
MOVL C00394 V=800.0 PL=0
MOVL C00395 V=800.0 PL=0
MOVL C00396 V=800.0 PL=0
MOVL C00397 V=800.0 PL=0
MOVL C00398 V=800.0 PL=0
MOVL C00399 V=800.0 PL=0
MOVL C00400 V=800.0 PL=0
MOVL C00401 V=800.0 PL=0
MOVL C00402 V=800.0 PL=0
MOVL C00403 V=800.0 PL=0
MOVL C00404 V=800.0 PL=0
MOVL C00405 V=800.0 PL=0
MOVL C00406 V=800.0 PL=0
MOVL C00407 V=800.0 PL=0
MOVL C00408 V=800.0 PL=0
MOVL C00409 V=800.0 PL=0
MOVL C00410 V=800.0 PL=0
MOVL C00411 V=800.0 PL=0
MOVL C00412 V=800.0 PL=0
MOVL C00413 V=800.0 PL=0
MOVL C00414 V=800.0 PL=0
MOVL C00415 V=800.0 PL=0
MOVL C00416 V=800.0 PL=0
MOVL C00417 V=800.0 PL=0
MOVL C00418 V=800.0 PL=0
MOVL C00419 V=800.0 PL=0
MOVL C00420 V=800.0 PL=0
MOVL C00421 V=800.0 PL=0
MOVL C00422 V=800.0 PL=0
MOVL C00423 V=800.0 PL=0
MOVL C00424 V=800.0 PL=0
MOVL C00425 V=800.0 PL=0
MOVL C00426 V=800.0 PL=0
MOVL C00427 V=800.0 PL=0
MOVL C00428 V=800.0 PL=0
MOVL C00429 V=800.0 PL=0
MOVL C00430 V=800.0 PL=0
MOVL C00431 V=800.0 PL=0
MOVL C00432 V=800.0 PL=0
MOVL C00433 V=800.0 PL=0
MOVL C00434 V=800.0 PL=0
MOVL C00435 V=800.0 PL=0
MOVL C00436 V=800.0 PL=0
MOVL C00437 V=800.0 PL=0
MOVL C00438 V=800.0 PL=0
MOVL C00439 V=800.0 PL=0
MOVL C00440 V=800.0 PL=0
MOVL C00441 V=800.0 PL=0
MOVL C00442 V=800.0 PL=0
MOVL C00443 V=800.0 PL=0
MOVL C00444 V=800.0 PL=0
MOVL C00445 V=800.0 PL=0
MOVL C00446 V=800.0 PL=0
MOVL C00447 V=800.0 PL=0
MOVL C00448 V=800.0 PL=0
MOVL C00449 V=800.0 PL=0
MOVL C00450 V=800.0 PL=0
MOVL C00451 V=800.0 PL=0
MOVL C00452 V=800.0 PL=0
MOVL C00453 V=800.0 PL=0
MOVL C00454 V=800.0 PL=0
MOVL C00455 V=800.0 PL=0
MOVL C00456 V=800.0 PL=0
MOVL C00457 V=800.0 PL=0
MOVL C00458 V=800.0 PL=0
MOVL C00459 V=800.0 PL=0
MOVL C00460 V=800.0 PL=0
MOVL C00461 V=800.0 PL=0
MOVL C00462 V=800.0 PL=0
MOVL C00463 V=800.0 PL=0
MOVL C00464 V=800.0 PL=0
MOVL C00465 V=800.0 PL=0
MOVL C00466 V=800.0 PL=0
MOVL C00467 V=800.0 PL=0
MOVL C00468 V=800.0 PL=0
MOVL C00469 V=800.0 PL=0
MOVL C00470 V=800.0 PL=0
MOVL C00471 V=800.0 PL=0
MOVL C00472 V=800.0 PL=0
MOVL C00473 V=800.0 PL=0
MOVL C00474 V=800.0 PL=0
MOVL C00475 V=800.0 PL=0
MOVL C00476 V=800.0 PL=0
MOVL C00477 V=800.0 PL=0
MOVL C00478 V=800.0 PL=0
MOVL C00479 V=800.0 PL=0
MOVL C00480 V=800.0 PL=0
MOVL C00481 V=800.0 PL=0
MOVL C00482 V=800.0 PL=0
MOVL C00483 V=800.0 PL=0
MOVL C00484 V=800.0 PL=0
MOVL C00485 V=800.0 PL=0
MOVL C00486 V=800.0 PL=0
MOVL C00487 V=800.0 PL=0
MOVL C00488 V=800.0 PL=0
MOVL C00489 V=800.0 PL=0
MOVL C00490 V=800.0 PL=0
MOVL C00491 V=800.0 PL=0
MOVL C00492 V=800.0 PL=0
MOVL C00493 V=800.0 PL=0
MOVL C00494 V=800.0 PL=0
MOVL C00495 V=800.0 PL=0
MOVL C00496 V=800.0 PL=0
MOVL C00497 V=800.0 PL=0
MOVL C00498 V=800.0 PL=0
MOVL C00499 V=800.0 PL=0
MOVL C00500 V=800.0 PL=0
MOVL C00501 V=800.0 PL=0
MOVL C00502 V=800.0 PL=0
MOVL C00503 V=800.0 PL=0
MOVL C00504 V=800.0 PL=0
MOVL C00505 V=800.0 PL=0
MOVL C00506 V=800.0 PL=0
MOVL C00507 V=800.0 PL=0
MOVL C00508 V=800.0 PL=0
MOVL C00509 V=800.0 PL=0
MOVL C00510 V=800.0 PL=0
MOVL C00511 V=800.0 PL=0
MOVL C00512 V=800.0 PL=0
MOVL C00513 V=800.0 PL=0
MOVL C00514 V=800.0 PL=0
MOVL C00515 V=800.0 PL=0
MOVL C00516 V=800.0 PL=0
MOVL C00517 V=800.0 PL=0
MOVL C00518 V=800.0 PL=0
MOVL C00519 V=800.0 PL=0
MOVL C00520 V=800.0 PL=0
MOVL C00521 V=800.0 PL=0
MOVL C00522 V=800.0 PL=0
MOVL C00523 V=800.0 PL=0
MOVL C00524 V=800.0 PL=0
MOVL C00525 V=800.0 PL=0
MOVL C00526 V=800.0 PL=0
MOVL C00527 V=800.0 PL=0
MOVL C00528 V=800.0 PL=0
MOVL C00529 V=800.0 PL=0
MOVL C00530 V=800.0 PL=0
MOVL C00531 V=800.0 PL=0
MOVL C00532 V=800.0 PL=0
MOVL C00533 V=800.0 PL=0
MOVL C00534 V=800.0 PL=0
MOVL C00535 V=800.0 PL=0
MOVL C00536 V=800.0 PL=0
MOVL C00537 V=800.0 PL=0
MOVL C00538 V=800.0 PL=0
MOVL C00539 V=800.0 PL=0
MOVL C00540 V=800.0 PL=0
MOVL C00541 V=800.0 PL=0
MOVL C00542 V=800.0 PL=0
MOVL C00543 V=800.0 PL=0
MOVL C00544 V=800.0 PL=0
MOVL C00545 V=800.0 PL=0
MOVL C00546 V=800.0 PL=0
MOVL C00547 V=800.0 PL=0
MOVL C00548 V=800.0 PL=0
MOVL C00549 V=800.0 PL=0
MOVL C00550 V=800.0 PL=0
MOVL C00551 V=800.0 PL=0
MOVL C00552 V=800.0 PL=0
MOVL C00553 V=800.0 PL=0
MOVL C00554 V=800.0 PL=0
MOVL C00555 V=800.0 PL=0
MOVL C00556 V=800.0 PL=0
MOVL C00557 V=800.0 PL=0
MOVL C00558 V=800.0 PL=0
MOVL C00559 V=800.0 PL=0
MOVL C00560 V=800.0 PL=0
MOVL C00561 V=800.0 PL=0
MOVL C00562 V=800.0 PL=0
MOVL C00563 V=800.0 PL=0
MOVL C00564 V=800.0 PL=0
MOVL C00565 V=800.0 PL=0
MOVL C00566 V=800.0 PL=0
MOVL C00567 V=800.0 PL=0
MOVL C00568 V=800.0 PL=0
MOVL C00569 V=800.0 PL=0
MOVL C00570 V=800.0 PL=0
MOVL C00571 V=800.0 PL=0
MOVL C00572 V=800.0 PL=0
MOVL C00573 V=800.0 PL=0
MOVL C00574 V=800.0 PL=0
MOVL C00575 V=800.0 PL=0
MOVL C00576 V=800.0 PL=0
MOVL C00577 V=800.0 PL=0
MOVL C00578 V=800.0 PL=0
MOVL C00579 V=800.0 PL=0
MOVL C00580 V=800.0 PL=0
MOVL C00581 V=800.0 PL=0
MOVL C00582 V=800.0 PL=0
MOVL C00583 V=800.0 PL=0
MOVL C00584 V=800.0 PL=0
MOVL C00585 V=800.0 PL=0
MOVL C00586 V=800.0 PL=0
MOVL C00587 V=800.0 PL=0
MOVL C00588 V=800.0 PL=0
MOVL C00589 V=800.0 PL=0
MOVL C00590 V=800.0 PL=0
MOVL C00591 V=800.0 PL=0
MOVL C00592 V=800.0 PL=0
MOVL C00593 V=800.0 PL=0
MOVL C00594 V=800.0 PL=0
MOVL C00595 V=800.0 PL=0
MOVL C00596 V=800.0 PL=0
MOVL C00597 V=800.0 PL=0
MOVL C00598 V=800.0 PL=0
MOVL C00599 V=800.0 PL=0
MOVL C00600 V=800.0 PL=0
MOVL C00601 V=800.0 PL=0
MOVL C00602 V=800.0 PL=0
MOVL C00603 V=800.0 PL=0
MOVL C00604 V=800.0 PL=0
MOVL C00605 V=800.0 PL=0
MOVL C00606 V=800.0 PL=0
MOVL C00607 V=800.0 PL=0
MOVL C00608 V=800.0 PL=0
MOVL C00609 V=800.0 PL=0
MOVL C00610 V=800.0 PL=0
MOVL C00611 V=800.0 PL=0
MOVL C00612 V=800.0 PL=0
MOVL C00613 V=800.0 PL=0
MOVL C00614 V=800.0 PL=0
MOVL C00615 V=800.0 PL=0
MOVL C00616 V=800.0 PL=0
MOVL C00617 V=800.0 PL=0
MOVL C00618 V=800.0 PL=0
MOVL C00619 V=800.0 PL=0
MOVL C00620 V=800.0 PL=0
MOVL C00621 V=800.0 PL=0
MOVL C00622 V=800.0 PL=0
MOVL C00623 V=800.0 PL=0
MOVL C00624 V=800.0 PL=0
MOVL C00625 V=800.0 PL=0
MOVL C00626 V=800.0 PL=0
MOVL C00627 V=800.0 PL=0
MOVL C00628 V=800.0 PL=0
MOVL C00629 V=800.0 PL=0
MOVL C00630 V=800.0 PL=0
MOVL C00631 V=800.0 PL=0
MOVL C00632 V=800.0 PL=0
MOVL C00633 V=800.0 PL=0
MOVL C00634 V=800.0 PL=0
MOVL C00635 V=800.0 PL=0
MOVL C00636 V=800.0 PL=0
MOVL C00637 V=800.0 PL=0
MOVL C00638 V=800.0 PL=0
MOVL C00639 V=800.0 PL=0
MOVL C00640 V=800.0 PL=0
MOVL C00641 V=800.0 PL=0
MOVL C00642 V=800.0 PL=0
MOVL C00643 V=800.0 PL=0
MOVL C00644 V=800.0 PL=0
MOVL C00645 V=800.0 PL=0
MOVL C00646 V=800.0 PL=0
MOVL C00647 V=800.0 PL=0
MOVL C00648 V=800.0 PL=0
MOVL C00649 V=800.0 PL=0
MOVL C00650 V=800.0 PL=0
MOVL C00651 V=800.0 PL=0
MOVL C00652 V=800.0 PL=0
MOVL C00653 V=800.0 PL=0
MOVL C00654 V=800.0 PL=0
MOVL C00655 V=800.0 PL=0
MOVL C00656 V=800.0 PL=0
MOVL C00657 V=800.0 PL=0
MOVL C00658 V=800.0 PL=0
MOVL C00659 V=800.0 PL=0
MOVL C00660 V=800.0 PL=0
MOVL C00661 V=800.0 PL=0
MOVL C00662 V=800.0 PL=0
MOVL C00663 V=800.0 PL=0
MOVL C00664 V=800.0 PL=0
MOVL C00665 V=800.0 PL=0
MOVL C00666 V=800.0 PL=0
MOVL C00667 V=800.0 PL=0
MOVL C00668 V=800.0 PL=0
MOVL C00669 V=800.0 PL=0
MOVL C00670 V=800.0 PL=0
MOVL C00671 V=800.0 PL=0
MOVL C00672 V=800.0 PL=0
MOVL C00673 V=800.0 PL=0
MOVL C00674 V=800.0 PL=0
MOVL C00675 V=800.0 PL=0
MOVL C00676 V=800.0 PL=0
MOVL C00677 V=800.0 PL=0
MOVL C00678 V=800.0 PL=0
MOVL C00679 V=800.0 PL=0
MOVL C00680 V=800.0 PL=0
MOVL C00681 V=800.0 PL=0
MOVL C00682 V=800.0 PL=0
MOVL C00683 V=800.0 PL=0
MOVL C00684 V=800.0 PL=0
MOVL C00685 V=800.0 PL=0
MOVL C00686 V=800.0 PL=0
MOVL C00687 V=800.0 PL=0
MOVL C00688 V=800.0 PL=0
MOVL C00689 V=800.0 PL=0
MOVL C00690 V=800.0 PL=0
MOVL C00691 V=800.0 PL=0
MOVL C00692 V=800.0 PL=0
MOVL C00693 V=800.0 PL=0
MOVL C00694 V=800.0 PL=0
MOVL C00695 V=800.0 PL=0
MOVL C00696 V=800.0 PL=0
MOVL C00697 V=800.0 PL=0
MOVL C00698 V=800.0 PL=0
MOVL C00699 V=800.0 PL=0
MOVL C00700 V=800.0 PL=0
MOVL C00701 V=800.0 PL=0
MOVL C00702 V=800.0 PL=0
MOVL C00703 V=800.0 PL=0
MOVL C00704 V=800.0 PL=0
MOVL C00705 V=800.0 PL=0
MOVL C00706 V=800.0 PL=0
MOVL C00707 V=800.0 PL=0
MOVL C00708 V=800.0 PL=0
MOVL C00709 V=800.0 PL=0
MOVL C00710 V=800.0 PL=0
MOVL C00711 V=800.0 PL=0
MOVL C00712 V=800.0 PL=0
MOVL C00713 V=800.0 PL=0
MOVL C00714 V=800.0 PL=0
MOVL C00715 V=800.0 PL=0
MOVL C00716 V=800.0 PL=0
MOVL C00717 V=800.0 PL=0
MOVL C00718 V=800.0 PL=0
MOVL C00719 V=800.0 PL=0
MOVL C00720 V=800.0 PL=0
MOVL C00721 V=800.0 PL=0
MOVL C00722 V=800.0 PL=0
MOVL C00723 V=800.0 PL=0
MOVL C00724 V=800.0 PL=0
MOVL C00725 V=800.0 PL=0
MOVL C00726 V=800.0 PL=0
MOVL C00727 V=800.0 PL=0
MOVL C00728 V=800.0 PL=0
MOVL C00729 V=800.0 PL=0
MOVL C00730 V=800.0 PL=0
MOVL C00731 V=800.0 PL=0
MOVL C00732 V=800.0 PL=0
MOVL C00733 V=800.0 PL=0
MOVL C00734 V=800.0 PL=0
MOVL C00735 V=800.0 PL=0
MOVL C00736 V=800.0 PL=0
MOVL C00737 V=800.0 PL=0
MOVL C00738 V=800.0 PL=0
MOVL C00739 V=800.0 PL=0
MOVL C00740 V=800.0 PL=0
MOVL C00741 V=800.0 PL=0
MOVL C00742 V=800.0 PL=0
MOVL C00743 V=800.0 PL=0
MOVL C00744 V=800.0 PL=0
MOVL C00745 V=800.0 PL=0
MOVL C00746 V=800.0 PL=0
MOVL C00747 V=800.0 PL=0
MOVL C00748 V=800.0 PL=0
MOVL C00749 V=800.0 PL=0
MOVL C00750 V=800.0 PL=0
MOVL C00751 V=800.0 PL=0
MOVL C00752 V=800.0 PL=0
MOVL C00753 V=800.0 PL=0
MOVL C00754 V=800.0 PL=0
MOVL C00755 V=800.0 PL=0
MOVL C00756 V=800.0 PL=0
MOVL C00757 V=800.0 PL=0
MOVL C00758 V=800.0 PL=0
MOVL C00759 V=800.0 PL=0
MOVL C00760 V=800.0 PL=0
MOVL C00761 V=800.0 PL=0
MOVL C00762 V=800.0 PL=0
MOVL C00763 V=800.0 PL=0
MOVL C00764 V=800.0 PL=0
MOVL C00765 V=800.0 PL=0
MOVL C00766 V=800.0 PL=0
MOVL C00767 V=800.0 PL=0
MOVL C00768 V=800.0 PL=0
MOVL C00769 V=800.0 PL=0
MOVL C00770 V=800.0 PL=0
MOVL C00771 V=800.0 PL=0
MOVL C00772 V=800.0 PL=0
MOVL C00773 V=800.0 PL=0
MOVL C00774 V=800.0 PL=0
MOVL C00775 V=800.0 PL=0
MOVL C00776 V=800.0 PL=0
MOVL C00777 V=800.0 PL=0
MOVL C00778 V=800.0 PL=0
MOVL C00779 V=800.0 PL=0
MOVL C00780 V=800.0 PL=0
MOVL C00781 V=800.0 PL=0
MOVL C00782 V=800.0 PL=0
MOVL C00783 V=800.0 PL=0
MOVL C00784 V=800.0 PL=0
MOVL C00785 V=800.0 PL=0
MOVL C00786 V=800.0 PL=0
MOVL C00787 V=800.0 PL=0
MOVL C00788 V=800.0 PL=0
MOVL C00789 V=800.0 PL=0
MOVL C00790 V=800.0 PL=0
MOVL C00791 V=800.0 PL=0
MOVL C00792 V=800.0 PL=0
MOVL C00793 V=800.0 PL=0
MOVL C00794 V=800.0 PL=0
MOVL C00795 V=800.0 PL=0
MOVL C00796 V=800.0 PL=0
MOVL C00797 V=800.0 PL=0
MOVL C00798 V=800.0 PL=0
MOVL C00799 V=800.0 PL=0
MOVL C00800 V=800.0 PL=0
MOVL C00801 V=800.0 PL=0
MOVL C00802 V=800.0 PL=0
MOVL C00803 V=800.0 PL=0
MOVL C00804 V=800.0 PL=0
MOVL C00805 V=800.0 PL=0
MOVL C00806 V=800.0 PL=0
MOVL C00807 V=800.0 PL=0
MOVL C00808 V=800.0 PL=0
MOVL C00809 V=800.0 PL=0
MOVL C00810 V=800.0 PL=0
MOVL C00811 V=800.0 PL=0
MOVL C00812 V=800.0 PL=0
MOVL C00813 V=800.0 PL=0
MOVL C00814 V=800.0 PL=0
MOVL C00815 V=800.0 PL=0
MOVL C00816 V=800.0 PL=0
MOVL C00817 V=800.0 PL=0
MOVL C00818 V=800.0 PL=0
MOVL C00819 V=800.0 PL=0
MOVL C00820 V=800.0 PL=0
MOVL C00821 V=800.0 PL=0
MOVL C00822 V=800.0 PL=0
MOVL C00823 V=800.0 PL=0
MOVL C00824 V=800.0 PL=0
MOVL C00825 V=800.0 PL=0
MOVL C00826 V=800.0 PL=0
MOVL C00827 V=800.0 PL=0
MOVL C00828 V=800.0 PL=0
MOVL C00829 V=800.0 PL=0
MOVL C00830 V=800.0 PL=0
MOVL C00831 V=800.0 PL=0
MOVL C00832 V=800.0 PL=0
MOVL C00833 V=800.0 PL=0
MOVL C00834 V=800.0 PL=0
MOVL C00835 V=800.0 PL=0
MOVL C00836 V=800.0 PL=0
MOVL C00837 V=800.0 PL=0
MOVL C00838 V=800.0 PL=0
MOVL C00839 V=800.0 PL=0
MOVL C00840 V=800.0 PL=0
MOVL C00841 V=800.0 PL=0
MOVL C00842 V=800.0 PL=0
MOVL C00843 V=800.0 PL=0
MOVL C00844 V=800.0 PL=0
MOVL C00845 V=800.0 PL=0
MOVL C00846 V=800.0 PL=0
MOVL C00847 V=800.0 PL=0
MOVL C00848 V=800.0 PL=0
MOVL C00849 V=800.0 PL=0
MOVL C00850 V=800.0 PL=0
MOVL C00851 V=800.0 PL=0
MOVL C00852 V=800.0 PL=0
MOVL C00853 V=800.0 PL=0
MOVL C00854 V=800.0 PL=0
MOVL C00855 V=800.0 PL=0
MOVL C00856 V=800.0 PL=0
MOVL C00857 V=800.0 PL=0
MOVL C00858 V=800.0 PL=0
MOVL C00859 V=800.0 PL=0
MOVL C00860 V=800.0 PL=0
MOVL C00861 V=800.0 PL=0
MOVL C00862 V=800.0 PL=0
MOVL C00863 V=800.0 PL=0
MOVL C00864 V=800.0 PL=0
MOVL C00865 V=800.0 PL=0
MOVL C00866 V=800.0 PL=0
MOVL C00867 V=800.0 PL=0
MOVL C00868 V=800.0 PL=0
MOVL C00869 V=800.0 PL=0
MOVL C00870 V=800.0 PL=0
MOVL C00871 V=800.0 PL=0
MOVL C00872 V=800.0 PL=0
MOVL C00873 V=800.0 PL=0
MOVL C00874 V=800.0 PL=0
MOVL C00875 V=800.0 PL=0
MOVL C00876 V=800.0 PL=0
MOVL C00877 V=800.0 PL=0
MOVL C00878 V=800.0 PL=0
MOVL C00879 V=800.0 PL=0
MOVL C00880 V=800.0 PL=0
MOVL C00881 V=800.0 PL=0
MOVL C00882 V=800.0 PL=0
MOVL C00883 V=800.0 PL=0
MOVL C00884 V=800.0 PL=0
MOVL C00885 V=800.0 PL=0
MOVL C00886 V=800.0 PL=0
MOVL C00887 V=800.0 PL=0
MOVL C00888 V=800.0 PL=0
MOVL C00889 V=800.0 PL=0
MOVL C00890 V=800.0 PL=0
MOVL C00891 V=800.0 PL=0
MOVL C00892 V=800.0 PL=0
MOVL C00893 V=800.0 PL=0
MOVL C00894 V=800.0 PL=0
MOVL C00895 V=800.0 PL=0
MOVL C00896 V=800.0 PL=0
MOVL C00897 V=800.0 PL=0
MOVL C00898 V=800.0 PL=0
MOVL C00899 V=800.0 PL=0
MOVL C00900 V=800.0 PL=0
MOVL C00901 V=800.0 PL=0
MOVL C00902 V=800.0 PL=0
MOVL C00903 V=800.0 PL=0
MOVL C00904 V=800.0 PL=0
MOVL C00905 V=800.0 PL=0
MOVL C00906 V=800.0 PL=0
MOVL C00907 V=800.0 PL=0
MOVL C00908 V=800.0 PL=0
MOVL C00909 V=800.0 PL=0
MOVL C00910 V=800.0 PL=0
MOVL C00911 V=800.0 PL=0
MOVL C00912 V=800.0 PL=0
MOVL C00913 V=800.0 PL=0
MOVL C00914 V=800.0 PL=0
MOVL C00915 V=800.0 PL=0
MOVL C00916 V=800.0 PL=0
MOVL C00917 V=800.0 PL=0
MOVL C00918 V=800.0 PL=0
MOVL C00919 V=800.0 PL=0
MOVL C00920 V=800.0 PL=0
MOVL C00921 V=800.0 PL=0
MOVL C00922 V=800.0 PL=0
MOVL C00923 V=800.0 PL=0
MOVL C00924 V=800.0 PL=0
MOVL C00925 V=800.0 PL=0
MOVL C00926 V=800.0 PL=0
MOVL C00927 V=800.0 PL=0
MOVL C00928 V=800.0 PL=0
MOVL C00929 V=800.0 PL=0
MOVL C00930 V=800.0 PL=0
MOVL C00931 V=800.0 PL=0
MOVL C00932 V=800.0 PL=0
MOVL C00933 V=800.0 PL=0
MOVL C00934 V=800.0 PL=0
MOVL C00935 V=800.0 PL=0
MOVL C00936 V=800.0 PL=0
MOVL C00937 V=800.0 PL=0
MOVL C00938 V=800.0 PL=0
MOVL C00939 V=800.0 PL=0
MOVL C00940 V=800.0 PL=0
MOVL C00941 V=800.0 PL=0
MOVL C00942 V=800.0 PL=0
MOVL C00943 V=800.0 PL=0
MOVL C00944 V=800.0 PL=0
MOVL C00945 V=800.0 PL=0
MOVL C00946 V=800.0 PL=0
MOVL C00947 V=800.0 PL=0
MOVL C00948 V=800.0 PL=0
MOVL C00949 V=800.0 PL=0
MOVL C00950 V=800.0 PL=0
MOVL C00951 V=800.0 PL=0
MOVL C00952 V=800.0 PL=0
MOVL C00953 V=800.0 PL=0
MOVL C00954 V=800.0 PL=0
MOVL C00955 V=800.0 PL=0
MOVL C00956 V=800.0 PL=0
MOVL C00957 V=800.0 PL=0
MOVL C00958 V=800.0 PL=0
MOVL C00959 V=800.0 PL=0
MOVL C00960 V=800.0 PL=0
MOVL C00961 V=800.0 PL=0
MOVL C00962 V=800.0 PL=0
MOVL C00963 V=800.0 PL=0
MOVL C00964 V=800.0 PL=0
MOVL C00965 V=800.0 PL=0
MOVL C00966 V=800.0 PL=0
MOVL C00967 V=800.0 PL=0
MOVL C00968 V=800.0 PL=0
MOVL C00969 V=800.0 PL=0
MOVL C00970 V=800.0 PL=0
MOVL C00971 V=800.0 PL=0
MOVL C00972 V=800.0 PL=0
MOVL C00973 V=800.0 PL=0
MOVL C00974 V=800.0 PL=0
MOVL C00975 V=800.0 PL=0
MOVL C00976 V=800.0 PL=0
MOVL C00977 V=800.0 PL=0
MOVL C00978 V=800.0 PL=0
MOVL C00979 V=800.0 PL=0
MOVL C00980 V=800.0 PL=0
MOVL C00981 V=800.0 PL=0
MOVL C00982 V=800.0 PL=0
MOVL C00983 V=800.0 PL=0
MOVL C00984 V=800.0 PL=0
MOVL C00985 V=800.0 PL=0
MOVL C00986 V=800.0 PL=0
MOVL C00987 V=800.0 PL=0
MOVL C00988 V=800.0 PL=0
MOVL C00989 V=800.0 PL=0
MOVL C00990 V=800.0 PL=0
MOVL C00991 V=800.0 PL=0
MOVL C00992 V=800.0 PL=0
MOVL C00993 V=800.0 PL=0
MOVL C00994 V=800.0 PL=0
MOVL C00995 V=800.0 PL=0
MOVL C00996 V=800.0 PL=0
MOVL C00997 V=800.0 PL=0
MOVL C00998 V=800.0 PL=0
MOVL C00999 V=800.0 PL=0
MOVL C01000 V=800.0 PL=0
MOVL C01001 V=800.0 PL=0
MOVL C01002 V=800.0 PL=0
MOVL C01003 V=800.0 PL=0
MOVL C01004 V=800.0 PL=0
MOVL C01005 V=800.0 PL=0
MOVL C01006 V=800.0 PL=0
MOVL C01007 V=800.0 PL=0
MOVL C01008 V=800.0 PL=0
MOVL C01009 V=800.0 PL=0
MOVL C01010 V=800.0 PL=0
MOVL C01011 V=800.0 PL=0
MOVL C01012 V=800.0 PL=0
MOVL C01013 V=800.0 PL=0
MOVL C01014 V=800.0 PL=0
MOVL C01015 V=800.0 PL=0
MOVL C01016 V=800.0 PL=0
MOVL C01017 V=800.0 PL=0
MOVL C01018 V=800.0 PL=0
MOVL C01019 V=800.0 PL=0
MOVL C01020 V=800.0 PL=0
MOVL C01021 V=800.0 PL=0
MOVL C01022 V=800.0 PL=0
MOVL C01023 V=800.0 PL=0
MOVL C01024 V=800.0 PL=0
MOVL C01025 V=800.0 PL=0
MOVL C01026 V=800.0 PL=0
MOVL C01027 V=800.0 PL=0
MOVL C01028 V=800.0 PL=0
MOVL C01029 V=800.0 PL=0
MOVL C01030 V=800.0 PL=0
MOVL C01031 V=800.0 PL=0
MOVL C01032 V=800.0 PL=0
MOVL C01033 V=800.0 PL=0
MOVL C01034 V=800.0 PL=0
MOVL C01035 V=800.0 PL=0
MOVL C01036 V=800.0 PL=0
MOVL C01037 V=800.0 PL=0
MOVL C01038 V=800.0 PL=0
MOVL C01039 V=800.0 PL=0
MOVL C01040 V=800.0 PL=0
MOVL C01041 V=800.0 PL=0
MOVL C01042 V=800.0 PL=0
MOVL C01043 V=800.0 PL=0
MOVL C01044 V=800.0 PL=0
MOVL C01045 V=800.0 PL=0
MOVL C01046 V=800.0 PL=0
MOVL C01047 V=800.0 PL=0
MOVL C01048 V=800.0 PL=0
MOVL C01049 V=800.0 PL=0
MOVL C01050 V=800.0 PL=0
MOVL C01051 V=800.0 PL=0
MOVL C01052 V=800.0 PL=0
MOVL C01053 V=800.0 PL=0
MOVL C01054 V=800.0 PL=0
MOVL C01055 V=800.0 PL=0
MOVL C01056 V=800.0 PL=0
MOVL C01057 V=800.0 PL=0
MOVL C01058 V=800.0 PL=0
MOVL C01059 V=800.0 PL=0
MOVL C01060 V=800.0 PL=0
MOVL C01061 V=800.0 PL=0
MOVL C01062 V=800.0 PL=0
MOVL C01063 V=800.0 PL=0
MOVL C01064 V=800.0 PL=0
MOVL C01065 V=800.0 PL=0
MOVL C01066 V=800.0 PL=0
MOVL C01067 V=800.0 PL=0
MOVL C01068 V=800.0 PL=0
MOVL C01069 V=800.0 PL=0
MOVL C01070 V=800.0 PL=0
MOVL C01071 V=800.0 PL=0
MOVL C01072 V=800.0 PL=0
MOVL C01073 V=800.0 PL=0
MOVL C01074 V=800.0 PL=0
MOVL C01075 V=800.0 PL=0
MOVL C01076 V=800.0 PL=0
MOVL C01077 V=800.0 PL=0
MOVL C01078 V=800.0 PL=0
MOVL C01079 V=800.0 PL=0
MOVL C01080 V=800.0 PL=0
MOVL C01081 V=800.0 PL=0
MOVL C01082 V=800.0 PL=0
MOVL C01083 V=800.0 PL=0
MOVL C01084 V=800.0 PL=0
MOVL C01085 V=800.0 PL=0
MOVL C01086 V=800.0 PL=0
MOVL C01087 V=800.0 PL=0
MOVL C01088 V=800.0 PL=0
MOVL C01089 V=800.0 PL=0
MOVL C01090 V=800.0 PL=0
MOVL C01091 V=800.0 PL=0
MOVL C01092 V=800.0 PL=0
MOVL C01093 V=800.0 PL=0
MOVL C01094 V=800.0 PL=0
MOVL C01095 V=800.0 PL=0
MOVL C01096 V=800.0 PL=0
MOVL C01097 V=800.0 PL=0
MOVL C01098 V=800.0 PL=0
MOVL C01099 V=800.0 PL=0
MOVL C01100 V=800.0 PL=0
MOVL C01101 V=800.0 PL=0
MOVL C01102 V=800.0 PL=0
MOVL C01103 V=800.0 PL=0
MOVL C01104 V=800.0 PL=0
MOVL C01105 V=800.0 PL=0
MOVL C01106 V=800.0 PL=0
MOVL C01107 V=800.0 PL=0
MOVL C01108 V=800.0 PL=0
MOVL C01109 V=800.0 PL=0
MOVL C01110 V=800.0 PL=0
MOVL C01111 V=800.0 PL=0
MOVL C01112 V=800.0 PL=0
MOVL C01113 V=800.0 PL=0
MOVL C01114 V=800.0 PL=0
MOVL C01115 V=800.0 PL=0
MOVL C01116 V=800.0 PL=0
MOVL C01117 V=800.0 PL=0
MOVL C01118 V=800.0 PL=0
MOVL C01119 V=800.0 PL=0
MOVL C01120 V=800.0 PL=0
MOVL C01121 V=800.0 PL=0
MOVL C01122 V=800.0 PL=0
MOVL C01123 V=800.0 PL=0
MOVL C01124 V=800.0 PL=0
MOVL C01125 V=800.0 PL=0
MOVL C01126 V=800.0 PL=0
MOVL C01127 V=800.0 PL=0
MOVL C01128 V=800.0 PL=0
MOVL C01129 V=800.0 PL=0
MOVL C01130 V=800.0 PL=0
MOVL C01131 V=800.0 PL=0
MOVL C01132 V=800.0 PL=0
MOVL C01133 V=800.0 PL=0
MOVL C01134 V=800.0 PL=0
MOVL C01135 V=800.0 PL=0
MOVL C01136 V=800.0 PL=0
MOVL C01137 V=800.0 PL=0
MOVL C01138 V=800.0 PL=0
MOVL C01139 V=800.0 PL=0
MOVL C01140 V=800.0 PL=0
MOVL C01141 V=800.0 PL=0
MOVL C01142 V=800.0 PL=0
MOVL C01143 V=800.0 PL=0
MOVL C01144 V=800.0 PL=0
MOVL C01145 V=800.0 PL=0
MOVL C01146 V=800.0 PL=0
MOVL C01147 V=800.0 PL=0
MOVL C01148 V=800.0 PL=0
MOVL C01149 V=800.0 PL=0
MOVL C01150 V=800.0 PL=0
MOVL C01151 V=800.0 PL=0
MOVL C01152 V=800.0 PL=0
MOVL C01153 V=800.0 PL=0
MOVL C01154 V=800.0 PL=0
MOVL C01155 V=800.0 PL=0
MOVL C01156 V=800.0 PL=0
MOVL C01157 V=800.0 PL=0
MOVL C01158 V=800.0 PL=0
MOVL C01159 V=800.0 PL=0
MOVL C01160 V=800.0 PL=0
MOVL C01161 V=800.0 PL=0
MOVL C01162 V=800.0 PL=0
MOVL C01163 V=800.0 PL=0
MOVL C01164 V=800.0 PL=0
MOVL C01165 V=800.0 PL=0
MOVL C01166 V=800.0 PL=0
MOVL C01167 V=800.0 PL=0
MOVL C01168 V=800.0 PL=0
MOVL C01169 V=800.0 PL=0
MOVL C01170 V=800.0 PL=0
MOVL C01171 V=800.0 PL=0
MOVL C01172 V=800.0 PL=0
MOVL C01173 V=800.0 PL=0
MOVL C01174 V=800.0 PL=0
MOVL C01175 V=800.0 PL=0
MOVL C01176 V=800.0 PL=0
MOVL C01177 V=800.0 PL=0
MOVL C01178 V=800.0 PL=0
MOVL C01179 V=800.0 PL=0
MOVL C01180 V=800.0 PL=0
MOVL C01181 V=800.0 PL=0
MOVL C01182 V=800.0 PL=0
MOVL C01183 V=800.0 PL=0
MOVL C01184 V=800.0 PL=0
MOVL C01185 V=800.0 PL=0
MOVL C01186 V=800.0 PL=0
MOVL C01187 V=800.0 PL=0
MOVL C01188 V=800.0 PL=0
MOVL C01189 V=800.0 PL=0
MOVL C01190 V=800.0 PL=0
MOVL C01191 V=800.0 PL=0
MOVL C01192 V=800.0 PL=0
MOVL C01193 V=800.0 PL=0
MOVL C01194 V=800.0 PL=0
MOVL C01195 V=800.0 PL=0
MOVL C01196 V=800.0 PL=0
MOVL C01197 V=800.0 PL=0
MOVL C01198 V=800.0 PL=0
MOVL C01199 V=800.0 PL=0
MOVL C01200 V=800.0 PL=0
MOVL C01201 V=800.0 PL=0
MOVL C01202 V=800.0 PL=0
MOVL C01203 V=800.0 PL=0
MOVL C01204 V=800.0 PL=0
MOVL C01205 V=800.0 PL=0
MOVL C01206 V=800.0 PL=0
MOVL C01207 V=800.0 PL=0
MOVL C01208 V=800.0 PL=0
MOVL C01209 V=800.0 PL=0
MOVL C01210 V=800.0 PL=0
MOVL C01211 V=800.0 PL=0
MOVL C01212 V=800.0 PL=0
MOVL C01213 V=800.0 PL=0
MOVL C01214 V=800.0 PL=0
MOVL C01215 V=800.0 PL=0
MOVL C01216 V=800.0 PL=0
MOVL C01217 V=800.0 PL=0
MOVL C01218 V=800.0 PL=0
MOVL C01219 V=800.0 PL=0
MOVL C01220 V=800.0 PL=0
MOVL C01221 V=800.0 PL=0
MOVL C01222 V=800.0 PL=0
MOVL C01223 V=800.0 PL=0
MOVL C01224 V=800.0 PL=0
MOVL C01225 V=800.0 PL=0
MOVL C01226 V=800.0 PL=0
MOVL C01227 V=800.0 PL=0
MOVL C01228 V=800.0 PL=0
MOVL C01229 V=800.0 PL=0
MOVL C01230 V=800.0 PL=0
MOVL C01231 V=800.0 PL=0
MOVL C01232 V=800.0 PL=0
MOVL C01233 V=800.0 PL=0
MOVL C01234 V=800.0 PL=0
MOVL C01235 V=800.0 PL=0
MOVL C01236 V=800.0 PL=0
MOVL C01237 V=800.0 PL=0
MOVL C01238 V=800.0 PL=0
MOVL C01239 V=800.0 PL=0
MOVL C01240 V=800.0 PL=0
MOVL C01241 V=800.0 PL=0
MOVL C01242 V=800.0 PL=0
MOVL C01243 V=800.0 PL=0
MOVL C01244 V=800.0 PL=0
MOVL C01245 V=800.0 PL=0
MOVL C01246 V=800.0 PL=0
MOVL C01247 V=800.0 PL=0
MOVL C01248 V=800.0 PL=0
MOVL C01249 V=800.0 PL=0
MOVL C01250 V=800.0 PL=0
MOVL C01251 V=800.0 PL=0
MOVL C01252 V=800.0 PL=0
MOVL C01253 V=800.0 PL=0
MOVL C01254 V=800.0 PL=0
MOVL C01255 V=800.0 PL=0
MOVL C01256 V=800.0 PL=0
MOVL C01257 V=800.0 PL=0
MOVL C01258 V=800.0 PL=0
MOVL C01259 V=800.0 PL=0
MOVL C01260 V=800.0 PL=0
MOVL C01261 V=800.0 PL=0
MOVL C01262 V=800.0 PL=0
MOVL C01263 V=800.0 PL=0
MOVL C01264 V=800.0 PL=0
MOVL C01265 V=800.0 PL=0
MOVL C01266 V=800.0 PL=0
MOVL C01267 V=800.0 PL=0
MOVL C01268 V=800.0 PL=0
MOVL C01269 V=800.0 PL=0
MOVL C01270 V=800.0 PL=0
MOVL C01271 V=800.0 PL=0
MOVL C01272 V=800.0 PL=0
MOVL C01273 V=800.0 PL=0
MOVL C01274 V=800.0 PL=0
MOVL C01275 V=800.0 PL=0
MOVL C01276 V=800.0 PL=0
MOVL C01277 V=800.0 PL=0
MOVL C01278 V=800.0 PL=0
MOVL C01279 V=800.0 PL=0
MOVL C01280 V=800.0 PL=0
MOVL C01281 V=800.0 PL=0
MOVL C01282 V=800.0 PL=0
MOVL C01283 V=800.0 PL=0
MOVL C01284 V=800.0 PL=0
MOVL C01285 V=800.0 PL=0
MOVL C01286 V=800.0 PL=0
MOVL C01287 V=800.0 PL=0
MOVL C01288 V=800.0 PL=0
MOVL C01289 V=800.0 PL=0
MOVL C01290 V=800.0 PL=0
MOVL C01291 V=800.0 PL=0
MOVL C01292 V=800.0 PL=0
MOVL C01293 V=800.0 PL=0
MOVL C01294 V=800.0 PL=0
MOVL C01295 V=800.0 PL=0
MOVL C01296 V=800.0 PL=0
MOVL C01297 V=800.0 PL=0
MOVL C01298 V=800.0 PL=0
MOVL C01299 V=800.0 PL=0
MOVL C01300 V=800.0 PL=0
MOVL C01301 V=800.0 PL=0
MOVL C01302 V=800.0 PL=0
MOVL C01303 V=800.0 PL=0
MOVL C01304 V=800.0 PL=0
MOVL C01305 V=800.0 PL=0
MOVL C01306 V=800.0 PL=0
MOVL C01307 V=800.0 PL=0
MOVL C01308 V=800.0 PL=0
MOVL C01309 V=800.0 PL=0
MOVL C01310 V=800.0 PL=0
MOVL C01311 V=800.0 PL=0
MOVL C01312 V=800.0 PL=0
MOVL C01313 V=800.0 PL=0
MOVL C01314 V=800.0 PL=0
MOVL C01315 V=800.0 PL=0
MOVL C01316 V=800.0 PL=0
MOVL C01317 V=800.0 PL=0
MOVL C01318 V=800.0 PL=0
MOVL C01319 V=800.0 PL=0
MOVL C01320 V=800.0 PL=0
MOVL C01321 V=800.0 PL=0
MOVL C01322 V=800.0 PL=0
MOVL C01323 V=800.0 PL=0
MOVL C01324 V=800.0 PL=0
MOVL C01325 V=800.0 PL=0
MOVL C01326 V=800.0 PL=0
MOVL C01327 V=800.0 PL=0
MOVL C01328 V=800.0 PL=0
MOVL C01329 V=800.0 PL=0
MOVL C01330 V=800.0 PL=0
MOVL C01331 V=800.0 PL=0
MOVL C01332 V=800.0 PL=0
MOVL C01333 V=800.0 PL=0
MOVL C01334 V=800.0 PL=0
MOVL C01335 V=800.0 PL=0
MOVL C01336 V=800.0 PL=0
MOVL C01337 V=800.0 PL=0
MOVL C01338 V=800.0 PL=0
MOVL C01339 V=800.0 PL=0
MOVL C01340 V=800.0 PL=0
MOVL C01341 V=800.0 PL=0
MOVL C01342 V=800.0 PL=0
MOVL C01343 V=800.0 PL=0
MOVL C01344 V=800.0 PL=0
MOVL C01345 V=800.0 PL=0
MOVL C01346 V=800.0 PL=0
MOVL C01347 V=800.0 PL=0
MOVL C01348 V=800.0 PL=0
MOVL C01349 V=800.0 PL=0
MOVL C01350 V=800.0 PL=0
MOVL C01351 V=800.0 PL=0
MOVL C01352 V=800.0 PL=0
MOVL C01353 V=800.0 PL=0
MOVL C01354 V=800.0 PL=0
MOVL C01355 V=800.0 PL=0
MOVL C01356 V=800.0 PL=0
MOVL C01357 V=800.0 PL=0
MOVL C01358 V=800.0 PL=0
MOVL C01359 V=800.0 PL=0
MOVL C01360 V=800.0 PL=0
MOVL C01361 V=800.0 PL=0
MOVL C01362 V=800.0 PL=0
MOVL C01363 V=800.0 PL=0
MOVL C01364 V=800.0 PL=0
MOVL C01365 V=800.0 PL=0
MOVL C01366 V=800.0 PL=0
MOVL C01367 V=800.0 PL=0
MOVL C01368 V=800.0 PL=0
MOVL C01369 V=800.0 PL=0
MOVL C01370 V=800.0 PL=0
MOVL C01371 V=800.0 PL=0
MOVL C01372 V=800.0 PL=0
MOVL C01373 V=800.0 PL=0
MOVL C01374 V=800.0 PL=0
MOVL C01375 V=800.0 PL=0
MOVL C01376 V=800.0 PL=0
MOVL C01377 V=800.0 PL=0
MOVL C01378 V=800.0 PL=0
MOVL C01379 V=800.0 PL=0
MOVL C01380 V=800.0 PL=0
MOVL C01381 V=800.0 PL=0
MOVL C01382 V=800.0 PL=0
MOVL C01383 V=800.0 PL=0
MOVL C01384 V=800.0 PL=0
MOVL C01385 V=800.0 PL=0
MOVL C01386 V=800.0 PL=0
MOVL C01387 V=800.0 PL=0
MOVL C01388 V=800.0 PL=0
MOVL C01389 V=800.0 PL=0
MOVL C01390 V=800.0 PL=0
MOVL C01391 V=800.0 PL=0
MOVL C01392 V=800.0 PL=0
MOVL C01393 V=800.0 PL=0
MOVL C01394 V=800.0 PL=0
MOVL C01395 V=800.0 PL=0
MOVL C01396 V=800.0 PL=0
MOVL C01397 V=800.0 PL=0
MOVL C01398 V=800.0 PL=0
MOVL C01399 V=800.0 PL=0
MOVL C01400 V=800.0 PL=0
MOVL C01401 V=800.0 PL=0
MOVL C01402 V=800.0 PL=0
MOVL C01403 V=800.0 PL=0
MOVL C01404 V=800.0 PL=0
MOVL C01405 V=800.0 PL=0
MOVL C01406 V=800.0 PL=0
MOVL C01407 V=800.0 PL=0
MOVL C01408 V=800.0 PL=0
MOVL C01409 V=800.0 PL=0
MOVL C01410 V=800.0 PL=0
MOVL C01411 V=800.0 PL=0
MOVL C01412 V=800.0 PL=0
MOVL C01413 V=800.0 PL=0
MOVL C01414 V=800.0 PL=0
MOVL C01415 V=800.0 PL=0
MOVL C01416 V=800.0 PL=0
MOVL C01417 V=800.0 PL=0
MOVL C01418 V=800.0 PL=0
MOVL C01419 V=800.0 PL=0
MOVL C01420 V=800.0 PL=0
MOVL C01421 V=800.0 PL=0
MOVL C01422 V=800.0 PL=0
MOVL C01423 V=800.0 PL=0
MOVL C01424 V=800.0 PL=0
MOVL C01425 V=800.0 PL=0
MOVL C01426 V=800.0 PL=0
MOVL C01427 V=800.0 PL=0
MOVL C01428 V=800.0 PL=0
MOVL C01429 V=800.0 PL=0
MOVL C01430 V=800.0 PL=0
MOVL C01431 V=800.0 PL=0
MOVL C01432 V=800.0 PL=0
MOVL C01433 V=800.0 PL=0
MOVL C01434 V=800.0 PL=0
MOVL C01435 V=800.0 PL=0
MOVL C01436 V=800.0 PL=0
MOVL C01437 V=800.0 PL=0
MOVL C01438 V=800.0 PL=0
MOVL C01439 V=800.0 PL=0
MOVL C01440 V=800.0 PL=0
MOVL C01441 V=800.0 PL=0
MOVL C01442 V=800.0 PL=0
MOVL C01443 V=800.0 PL=0
MOVL C01444 V=800.0 PL=0
MOVL C01445 V=800.0 PL=0
MOVL C01446 V=800.0 PL=0
MOVL C01447 V=800.0 PL=0
MOVL C01448 V=800.0 PL=0
MOVL C01449 V=800.0 PL=0
MOVL C01450 V=800.0 PL=0
MOVL C01451 V=800.0 PL=0
MOVL C01452 V=800.0 PL=0
MOVL C01453 V=800.0 PL=0
MOVL C01454 V=800.0 PL=0
MOVL C01455 V=800.0 PL=0
MOVL C01456 V=800.0 PL=0
MOVL C01457 V=800.0 PL=0
MOVL C01458 V=800.0 PL=0
MOVL C01459 V=800.0 PL=0
MOVL C01460 V=800.0 PL=0
MOVL C01461 V=800.0 PL=0
MOVL C01462 V=800.0 PL=0
MOVL C01463 V=800.0 PL=0
MOVL C01464 V=800.0 PL=0
MOVL C01465 V=800.0 PL=0
MOVL C01466 V=800.0 PL=0
MOVL C01467 V=800.0 PL=0
MOVL C01468 V=800.0 PL=0
MOVL C01469 V=800.0 PL=0
MOVL C01470 V=800.0 PL=0
MOVL C01471 V=800.0 PL=0
MOVL C01472 V=800.0 PL=0
MOVL C01473 V=800.0 PL=0
MOVL C01474 V=800.0 PL=0
MOVL C01475 V=800.0 PL=0
MOVL C01476 V=800.0 PL=0
MOVL C01477 V=800.0 PL=0
MOVL C01478 V=800.0 PL=0
MOVL C01479 V=800.0 PL=0
MOVL C01480 V=800.0 PL=0
MOVL C01481 V=800.0 PL=0
MOVL C01482 V=800.0 PL=0
MOVL C01483 V=800.0 PL=0
MOVL C01484 V=800.0 PL=0
MOVL C01485 V=800.0 PL=0
MOVL C01486 V=800.0 PL=0
MOVL C01487 V=800.0 PL=0
MOVL C01488 V=800.0 PL=0
MOVL C01489 V=800.0 PL=0
MOVL C01490 V=800.0 PL=0
MOVL C01491 V=800.0 PL=0
MOVL C01492 V=800.0 PL=0
MOVL C01493 V=800.0 PL=0
MOVL C01494 V=800.0 PL=0
MOVL C01495 V=800.0 PL=0
MOVL C01496 V=800.0 PL=0
MOVL C01497 V=800.0 PL=0
MOVL C01498 V=800.0 PL=0
MOVL C01499 V=800.0 PL=0
MOVL C01500 V=800.0 PL=0
MOVL C01501 V=800.0 PL=0
MOVL C01502 V=800.0 PL=0
MOVL C01503 V=800.0 PL=0
MOVL C01504 V=800.0 PL=0
MOVL C01505 V=800.0 PL=0
MOVL C01506 V=800.0 PL=0
MOVL C01507 V=800.0 PL=0
MOVL C01508 V=800.0 PL=0
MOVL C01509 V=800.0 PL=0
MOVL C01510 V=800.0 PL=0
MOVL C01511 V=800.0 PL=0
MOVL C01512 V=800.0 PL=0
MOVL C01513 V=800.0 PL=0
MOVL C01514 V=800.0 PL=0
MOVL C01515 V=800.0 PL=0
MOVL C01516 V=800.0 PL=0
MOVL C01517 V=800.0 PL=0
MOVL C01518 V=800.0 PL=0
MOVL C01519 V=800.0 PL=0
MOVL C01520 V=800.0 PL=0
MOVL C01521 V=800.0 PL=0
MOVL C01522 V=800.0 PL=0
MOVL C01523 V=800.0 PL=0
MOVL C01524 V=800.0 PL=0
MOVL C01525 V=800.0 PL=0
MOVL C01526 V=800.0 PL=0
MOVL C01527 V=800.0 PL=0
MOVL C01528 V=800.0 PL=0
MOVL C01529 V=800.0 PL=0
MOVL C01530 V=800.0 PL=0
MOVL C01531 V=800.0 PL=0
MOVL C01532 V=800.0 PL=0
MOVL C01533 V=800.0 PL=0
MOVL C01534 V=800.0 PL=0
MOVL C01535 V=800.0 PL=0
MOVL C01536 V=800.0 PL=0
MOVL C01537 V=800.0 PL=0
MOVL C01538 V=800.0 PL=0
MOVL C01539 V=800.0 PL=0
MOVL C01540 V=800.0 PL=0
MOVL C01541 V=800.0 PL=0
MOVL C01542 V=800.0 PL=0
MOVL C01543 V=800.0 PL=0
MOVL C01544 V=800.0 PL=0
MOVL C01545 V=800.0 PL=0
MOVL C01546 V=800.0 PL=0
MOVL C01547 V=800.0 PL=0
MOVL C01548 V=800.0 PL=0
MOVL C01549 V=800.0 PL=0
MOVL C01550 V=800.0 PL=0
MOVL C01551 V=800.0 PL=0
MOVL C01552 V=800.0 PL=0
MOVL C01553 V=800.0 PL=0
MOVL C01554 V=800.0 PL=0
MOVL C01555 V=800.0 PL=0
MOVL C01556 V=800.0 PL=0
MOVL C01557 V=800.0 PL=0
MOVL C01558 V=800.0 PL=0
MOVL C01559 V=800.0 PL=0
MOVL C01560 V=800.0 PL=0
MOVL C01561 V=800.0 PL=0
MOVL C01562 V=800.0 PL=0
MOVL C01563 V=800.0 PL=0
MOVL C01564 V=800.0 PL=0
MOVL C01565 V=800.0 PL=0
MOVL C01566 V=800.0 PL=0
MOVL C01567 V=800.0 PL=0
MOVL C01568 V=800.0 PL=0
MOVL C01569 V=800.0 PL=0
MOVL C01570 V=800.0 PL=0
MOVL C01571 V=800.0 PL=0
MOVL C01572 V=800.0 PL=0
MOVL C01573 V=800.0 PL=0
MOVL C01574 V=800.0 PL=0
MOVL C01575 V=800.0 PL=0
MOVL C01576 V=800.0 PL=0
MOVL C01577 V=800.0 PL=0
MOVL C01578 V=800.0 PL=0
MOVL C01579 V=800.0 PL=0
MOVL C01580 V=800.0 PL=0
MOVL C01581 V=800.0 PL=0
MOVL C01582 V=800.0 PL=0
MOVL C01583 V=800.0 PL=0
MOVL C01584 V=800.0 PL=0
MOVL C01585 V=800.0 PL=0
MOVL C01586 V=800.0 PL=0
MOVL C01587 V=800.0 PL=0
MOVL C01588 V=800.0 PL=0
MOVL C01589 V=800.0 PL=0
MOVL C01590 V=800.0 PL=0
MOVL C01591 V=800.0 PL=0
MOVL C01592 V=800.0 PL=0
MOVL C01593 V=800.0 PL=0
MOVL C01594 V=800.0 PL=0
MOVL C01595 V=800.0 PL=0
MOVL C01596 V=800.0 PL=0
MOVL C01597 V=800.0 PL=0
MOVL C01598 V=800.0 PL=0
MOVL C01599 V=800.0 PL=0
MOVL C01600 V=800.0 PL=0
MOVL C01601 V=800.0 PL=0
MOVL C01602 V=800.0 PL=0
MOVL C01603 V=800.0 PL=0
MOVL C01604 V=800.0 PL=0
MOVL C01605 V=800.0 PL=0
MOVL C01606 V=800.0 PL=0
MOVL C01607 V=800.0 PL=0
MOVL C01608 V=800.0 PL=0
MOVL C01609 V=800.0 PL=0
MOVL C01610 V=800.0 PL=0
MOVL C01611 V=800.0 PL=0
MOVL C01612 V=800.0 PL=0
MOVL C01613 V=800.0 PL=0
MOVL C01614 V=800.0 PL=0
MOVL C01615 V=800.0 PL=0
MOVL C01616 V=800.0 PL=0
MOVL C01617 V=800.0 PL=0
MOVL C01618 V=800.0 PL=0
MOVL C01619 V=800.0 PL=0
MOVL C01620 V=800.0 PL=0
MOVL C01621 V=800.0 PL=0
MOVL C01622 V=800.0 PL=0
MOVL C01623 V=800.0 PL=0
MOVL C01624 V=800.0 PL=0
MOVL C01625 V=800.0 PL=0
MOVL C01626 V=800.0 PL=0
MOVL C01627 V=800.0 PL=0
MOVL C01628 V=800.0 PL=0
MOVL C01629 V=800.0 PL=0
MOVL C01630 V=800.0 PL=0
MOVL C01631 V=800.0 PL=0
MOVL C01632 V=800.0 PL=0
MOVL C01633 V=800.0 PL=0
MOVL C01634 V=800.0 PL=0
MOVL C01635 V=800.0 PL=0
MOVL C01636 V=800.0 PL=0
MOVL C01637 V=800.0 PL=0
MOVL C01638 V=800.0 PL=0
MOVL C01639 V=800.0 PL=0
MOVL C01640 V=800.0 PL=0
MOVL C01641 V=800.0 PL=0
MOVL C01642 V=800.0 PL=0
MOVL C01643 V=800.0 PL=0
MOVL C01644 V=800.0 PL=0
MOVL C01645 V=800.0 PL=0
MOVL C01646 V=800.0 PL=0
MOVL C01647 V=800.0 PL=0
MOVL C01648 V=800.0 PL=0
MOVL C01649 V=800.0 PL=0
MOVL C01650 V=800.0 PL=0
MOVL C01651 V=800.0 PL=0
MOVL C01652 V=800.0 PL=0
MOVL C01653 V=800.0 PL=0
MOVL C01654 V=800.0 PL=0
MOVL C01655 V=800.0 PL=0
MOVL C01656 V=800.0 PL=0
MOVL C01657 V=800.0 PL=0
MOVL C01658 V=800.0 PL=0
MOVL C01659 V=800.0 PL=0
MOVL C01660 V=800.0 PL=0
MOVL C01661 V=800.0 PL=0
MOVL C01662 V=800.0 PL=0
MOVL C01663 V=800.0 PL=0
MOVL C01664 V=800.0 PL=0
MOVL C01665 V=800.0 PL=0
MOVL C01666 V=800.0 PL=0
MOVL C01667 V=800.0 PL=0
MOVL C01668 V=800.0 PL=0
MOVL C01669 V=800.0 PL=0
MOVL C01670 V=800.0 PL=0
MOVL C01671 V=800.0 PL=0
MOVL C01672 V=800.0 PL=0
MOVL C01673 V=800.0 PL=0
MOVL C01674 V=800.0 PL=0
MOVL C01675 V=800.0 PL=0
MOVL C01676 V=800.0 PL=0
MOVL C01677 V=800.0 PL=0
MOVL C01678 V=800.0 PL=0
MOVL C01679 V=800.0 PL=0
MOVL C01680 V=800.0 PL=0
MOVL C01681 V=800.0 PL=0
MOVL C01682 V=800.0 PL=0
MOVL C01683 V=800.0 PL=0
MOVL C01684 V=800.0 PL=0
MOVL C01685 V=800.0 PL=0
MOVL C01686 V=800.0 PL=0
MOVL C01687 V=800.0 PL=0
MOVL C01688 V=800.0 PL=0
MOVL C01689 V=800.0 PL=0
MOVL C01690 V=800.0 PL=0
MOVL C01691 V=800.0 PL=0
MOVL C01692 V=800.0 PL=0
MOVL C01693 V=800.0 PL=0
MOVL C01694 V=800.0 PL=0
MOVL C01695 V=800.0 PL=0
MOVL C01696 V=800.0 PL=0
MOVL C01697 V=800.0 PL=0
MOVL C01698 V=800.0 PL=0
MOVL C01699 V=800.0 PL=0
MOVL C01700 V=800.0 PL=0
MOVL C01701 V=800.0 PL=0
MOVL C01702 V=800.0 PL=0
MOVL C01703 V=800.0 PL=0
MOVL C01704 V=800.0 PL=0
MOVL C01705 V=800.0 PL=0
MOVL C01706 V=800.0 PL=0
MOVL C01707 V=800.0 PL=0
MOVL C01708 V=800.0 PL=0
MOVL C01709 V=800.0 PL=0
MOVL C01710 V=800.0 PL=0
MOVL C01711 V=800.0 PL=0
MOVL C01712 V=800.0 PL=0
MOVL C01713 V=800.0 PL=0
MOVL C01714 V=800.0 PL=0
MOVL C01715 V=800.0 PL=0
MOVL C01716 V=800.0 PL=0
MOVL C01717 V=800.0 PL=0
MOVL C01718 V=800.0 PL=0
MOVL C01719 V=800.0 PL=0
MOVL C01720 V=800.0 PL=0
MOVL C01721 V=800.0 PL=0
MOVL C01722 V=800.0 PL=0
MOVL C01723 V=800.0 PL=0
MOVL C01724 V=800.0 PL=0
MOVL C01725 V=800.0 PL=0
MOVL C01726 V=800.0 PL=0
MOVL C01727 V=800.0 PL=0
MOVL C01728 V=800.0 PL=0
MOVL C01729 V=800.0 PL=0
MOVL C01730 V=800.0 PL=0
MOVL C01731 V=800.0 PL=0
MOVL C01732 V=800.0 PL=0
MOVL C01733 V=800.0 PL=0
MOVL C01734 V=800.0 PL=0
MOVL C01735 V=800.0 PL=0
MOVL C01736 V=800.0 PL=0
MOVL C01737 V=800.0 PL=0
MOVL C01738 V=800.0 PL=0
MOVL C01739 V=800.0 PL=0
MOVL C01740 V=800.0 PL=0
MOVL C01741 V=800.0 PL=0
MOVL C01742 V=800.0 PL=0
MOVL C01743 V=800.0 PL=0
MOVL C01744 V=800.0 PL=0
MOVL C01745 V=800.0 PL=0
MOVL C01746 V=800.0 PL=0
MOVL C01747 V=800.0 PL=0
MOVL C01748 V=800.0 PL=0
MOVL C01749 V=800.0 PL=0
MOVL C01750 V=800.0 PL=0
MOVL C01751 V=800.0 PL=0
MOVL C01752 V=800.0 PL=0
MOVL C01753 V=800.0 PL=0
MOVL C01754 V=800.0 PL=0
MOVL C01755 V=800.0 PL=0
MOVL C01756 V=800.0 PL=0
MOVL C01757 V=800.0 PL=0
MOVL C01758 V=800.0 PL=0
MOVL C01759 V=800.0 PL=0
MOVL C01760 V=800.0 PL=0
MOVL C01761 V=800.0 PL=0
MOVL C01762 V=800.0 PL=0
MOVL C01763 V=800.0 PL=0
MOVL C01764 V=800.0 PL=0
MOVL C01765 V=800.0 PL=0
MOVL C01766 V=800.0 PL=0
MOVL C01767 V=800.0 PL=0
MOVL C01768 V=800.0 PL=0
MOVL C01769 V=800.0 PL=0
MOVL C01770 V=800.0 PL=0
MOVL C01771 V=800.0 PL=0
MOVL C01772 V=800.0 PL=0
MOVL C01773 V=800.0 PL=0
MOVL C01774 V=800.0 PL=0
MOVL C01775 V=800.0 PL=0
MOVL C01776 V=800.0 PL=0
MOVL C01777 V=800.0 PL=0
MOVL C01778 V=800.0 PL=0
MOVL C01779 V=800.0 PL=0
MOVL C01780 V=800.0 PL=0
MOVL C01781 V=800.0 PL=0
MOVL C01782 V=800.0 PL=0
MOVL C01783 V=800.0 PL=0
MOVL C01784 V=800.0 PL=0
MOVL C01785 V=800.0 PL=0
MOVL C01786 V=800.0 PL=0
MOVL C01787 V=800.0 PL=0
MOVL C01788 V=800.0 PL=0
MOVL C01789 V=800.0 PL=0
MOVL C01790 V=800.0 PL=0
MOVL C01791 V=800.0 PL=0
MOVL C01792 V=800.0 PL=0
MOVL C01793 V=800.0 PL=0
MOVL C01794 V=800.0 PL=0
MOVL C01795 V=800.0 PL=0
MOVL C01796 V=800.0 PL=0
MOVL C01797 V=800.0 PL=0
MOVL C01798 V=800.0 PL=0
MOVL C01799 V=800.0 PL=0
MOVL C01800 V=800.0 PL=0
MOVL C01801 V=800.0 PL=0
MOVL C01802 V=800.0 PL=0
MOVL C01803 V=800.0 PL=0
MOVL C01804 V=800.0 PL=0
MOVL C01805 V=800.0 PL=0
MOVL C01806 V=800.0 PL=0
MOVL C01807 V=800.0 PL=0
MOVL C01808 V=800.0 PL=0
MOVL C01809 V=800.0 PL=0
MOVL C01810 V=800.0 PL=0
MOVL C01811 V=800.0 PL=0
MOVL C01812 V=800.0 PL=0
MOVL C01813 V=800.0 PL=0
MOVL C01814 V=800.0 PL=0
MOVL C01815 V=800.0 PL=0
MOVL C01816 V=800.0 PL=0
MOVL C01817 V=800.0 PL=0
MOVL C01818 V=800.0 PL=0
MOVL C01819 V=800.0 PL=0
MOVL C01820 V=800.0 PL=0
MOVL C01821 V=800.0 PL=0
MOVL C01822 V=800.0 PL=0
MOVL C01823 V=800.0 PL=0
MOVL C01824 V=800.0 PL=0
MOVL C01825 V=800.0 PL=0
MOVL C01826 V=800.0 PL=0
MOVL C01827 V=800.0 PL=0
MOVL C01828 V=800.0 PL=0
MOVL C01829 V=800.0 PL=0
MOVL C01830 V=800.0 PL=0
MOVL C01831 V=800.0 PL=0
MOVL C01832 V=800.0 PL=0
MOVL C01833 V=800.0 PL=0
MOVL C01834 V=800.0 PL=0
MOVL C01835 V=800.0 PL=0
MOVL C01836 V=800.0 PL=0
MOVL C01837 V=800.0 PL=0
MOVL C01838 V=800.0 PL=0
MOVL C01839 V=800.0 PL=0
MOVL C01840 V=800.0 PL=0
MOVL C01841 V=800.0 PL=0
MOVL C01842 V=800.0 PL=0
MOVL C01843 V=800.0 PL=0
MOVL C01844 V=800.0 PL=0
MOVL C01845 V=800.0 PL=0
MOVL C01846 V=800.0 PL=0
MOVL C01847 V=800.0 PL=0
MOVL C01848 V=800.0 PL=0
MOVL C01849 V=800.0 PL=0
MOVL C01850 V=800.0 PL=0
MOVL C01851 V=800.0 PL=0
MOVL C01852 V=800.0 PL=0
MOVL C01853 V=800.0 PL=0
MOVL C01854 V=800.0 PL=0
MOVL C01855 V=800.0 PL=0
MOVL C01856 V=800.0 PL=0
MOVL C01857 V=800.0 PL=0
MOVL C01858 V=800.0 PL=0
MOVL C01859 V=800.0 PL=0
MOVL C01860 V=800.0 PL=0
MOVL C01861 V=800.0 PL=0
MOVL C01862 V=800.0 PL=0
MOVL C01863 V=800.0 PL=0
MOVL C01864 V=800.0 PL=0
MOVL C01865 V=800.0 PL=0
MOVL C01866 V=800.0 PL=0
MOVL C01867 V=800.0 PL=0
MOVL C01868 V=800.0 PL=0
MOVL C01869 V=800.0 PL=0
MOVL C01870 V=800.0 PL=0
MOVL C01871 V=800.0 PL=0
MOVL C01872 V=800.0 PL=0
MOVL C01873 V=800.0 PL=0
MOVL C01874 V=800.0 PL=0
MOVL C01875 V=800.0 PL=0
MOVL C01876 V=800.0 PL=0
MOVL C01877 V=800.0 PL=0
MOVL C01878 V=800.0 PL=0
MOVL C01879 V=800.0 PL=0
MOVL C01880 V=800.0 PL=0
MOVL C01881 V=800.0 PL=0
MOVL C01882 V=800.0 PL=0
MOVL C01883 V=800.0 PL=0
MOVL C01884 V=800.0 PL=0
MOVL C01885 V=800.0 PL=0
MOVL C01886 V=800.0 PL=0
MOVL C01887 V=800.0 PL=0
MOVL C01888 V=800.0 PL=0
MOVL C01889 V=800.0 PL=0
MOVL C01890 V=800.0 PL=0
MOVL C01891 V=800.0 PL=0
MOVL C01892 V=800.0 PL=0
MOVL C01893 V=800.0 PL=0
MOVL C01894 V=800.0 PL=0
MOVL C01895 V=800.0 PL=0
MOVL C01896 V=800.0 PL=0
MOVL C01897 V=800.0 PL=0
MOVL C01898 V=800.0 PL=0
MOVL C01899 V=800.0 PL=0
MOVL C01900 V=800.0 PL=0
MOVL C01901 V=800.0 PL=0
MOVL C01902 V=800.0 PL=0
MOVL C01903 V=800.0 PL=0
MOVL C01904 V=800.0 PL=0
MOVL C01905 V=800.0 PL=0
MOVL C01906 V=800.0 PL=0
MOVL C01907 V=800.0 PL=0
MOVL C01908 V=800.0 PL=0
MOVL C01909 V=800.0 PL=0
MOVL C01910 V=800.0 PL=0
MOVL C01911 V=800.0 PL=0
MOVL C01912 V=800.0 PL=0
MOVL C01913 V=800.0 PL=0
MOVL C01914 V=800.0 PL=0
MOVL C01915 V=800.0 PL=0
MOVL C01916 V=800.0 PL=0
MOVL C01917 V=800.0 PL=0
MOVL C01918 V=800.0 PL=0
MOVL C01919 V=800.0 PL=0
MOVL C01920 V=800.0 PL=0
MOVL C01921 V=800.0 PL=0
MOVL C01922 V=800.0 PL=0
MOVL C01923 V=800.0 PL=0
MOVL C01924 V=800.0 PL=0
MOVL C01925 V=800.0 PL=0
MOVL C01926 V=800.0 PL=0
MOVL C01927 V=800.0 PL=0
MOVL C01928 V=800.0 PL=0
MOVL C01929 V=800.0 PL=0
MOVL C01930 V=800.0 PL=0
MOVL C01931 V=800.0 PL=0
MOVL C01932 V=800.0 PL=0
MOVL C01933 V=800.0 PL=0
MOVL C01934 V=800.0 PL=0
MOVL C01935 V=800.0 PL=0
MOVL C01936 V=800.0 PL=0
MOVL C01937 V=800.0 PL=0
MOVL C01938 V=800.0 PL=0
MOVL C01939 V=800.0 PL=0
MOVL C01940 V=800.0 PL=0
MOVL C01941 V=800.0 PL=0
MOVL C01942 V=800.0 PL=0
MOVL C01943 V=800.0 PL=0
MOVL C01944 V=800.0 PL=0
MOVL C01945 V=800.0 PL=0
MOVL C01946 V=800.0 PL=0
MOVL C01947 V=800.0 PL=0
MOVL C01948 V=800.0 PL=0
MOVL C01949 V=800.0 PL=0
MOVL C01950 V=800.0 PL=0
MOVL C01951 V=800.0 PL=0
MOVL C01952 V=800.0 PL=0
MOVL C01953 V=800.0 PL=0
MOVL C01954 V=800.0 PL=0
MOVL C01955 V=800.0 PL=0
MOVL C01956 V=800.0 PL=0
MOVL C01957 V=800.0 PL=0
MOVL C01958 V=800.0 PL=0
MOVL C01959 V=800.0 PL=0
MOVL C01960 V=800.0 PL=0
MOVL C01961 V=800.0 PL=0
MOVL C01962 V=800.0 PL=0
MOVL C01963 V=800.0 PL=0
MOVL C01964 V=800.0 PL=0
